      ;FOLD F324 = !E2164 & T8 + F324 ;%{SE}%MKUKATPVW %CVW_SPS %VBOASG %P 2:F324 = !E2164 & T8 + F324, 3: BOASG
         $FLAG[324] = NOT $IN[2164] AND $TIMER_FLAG[8] OR $FLAG[324]
      ;ENDFOLD
      ;FOLD -- RSK Sammelstoerung -- ;%{SE}%MKUKATPVW %CVW_COM %VCOMMENT %P 2:-- RSK Sammelstoerung --, 3: VW_COMMENT
      ;ENDFOLD
      ;FOLD F329 = F324 ;%{SE}%MKUKATPVW %CVW_SPS %VBOASG %P 2:F329 = F324, 3: BOASG
         $FLAG[329] = $FLAG[324]
      ;ENDFOLD
      ;FOLD A2164 = AUS ;%{SE}%MKUKATPVW %CVW_SPS %VBOASG %P 2:A2164 = AUS, 3: BOASG
         $OUT[2164] = FALSE
      ;ENDFOLD
      ;FOLD -- FRG Bewegung AUS -- ;%{SE}%MKUKATPVW %CVW_COM %VCOMMENT %P 2:-- FRG Bewegung AUS --, 3: VW_COMMENT
      ;ENDFOLD
      ;FOLD A2166 = AUS ;%{SE}%MKUKATPVW %CVW_SPS %VBOASG %P 2:A2166 = AUS, 3: BOASG
         $OUT[2166] = FALSE
      ;ENDFOLD
      ;FOLD -- FRG in Endlage halten ein -- ;%{SE}%MKUKATPVW %CVW_COM %VCOMMENT %P 2:-- FRG in Endlage halten ein --, 3: VW_COMMENT
      ;ENDFOLD
      ;FOLD A2165 = EIN ;%{SE}%MKUKATPVW %CVW_SPS %VBOASG %P 2:A2165 = EIN, 3: BOASG
         $OUT[2165] = TRUE
      ;ENDFOLD
      ;FOLD Schritt 154 = F324 & (E26 + E27) & A4039  ;%{SE}%MKUKATPVW %CVW_SPS %VST_CON %P 2:Schritt 154 = F324 & (E26 + E27) & A4039 , 3: ST_CON
         IF $FLAG[324] AND ($IN[26] OR $IN[27]) AND $OUT[4039] THEN
            PREVSTEP = $APP_INT[5]
            $APP_INT[5] = 154
         ENDIF
      ;ENDFOLD
      ;FOLD Schritt 158 = !F324 & E2164 & A4039  ;%{SE}%MKUKATPVW %CVW_SPS %VST_CON %P 2:Schritt 158 = !F324 & E2164 & A4039 , 3: ST_CON
         IF NOT $FLAG[324] AND $IN[2164] AND $OUT[4039] THEN
            PREVSTEP = $APP_INT[5]
            $APP_INT[5] = 158
         ENDIF
      ;ENDFOLD
   ;ENDFOLD
   ;FOLD SCHRITT 158 -- MS1 Reinigung (an Pneum. Schwenkeinheit MS1)-- ;%{P}%MKUKATPVW,%CSTEP,%VST_NR,%P 1:SCHRITT, 2:158, 3: MS1 Reinigung (an Pneum. Schwenkeinheit MS1)
      ;FOLD ;%{H}
         Case 158
      ;ENDFOLD
      ;FOLD -- Steuerluft EIN -- ;%{SE}%MKUKATPVW %CVW_COM %VCOMMENT %P 2:-- Steuerluft EIN --, 3: VW_COMMENT
      ;ENDFOLD
      ;FOLD A2161 = A4039 ;%{SE}%MKUKATPVW %CVW_SPS %VBOASG %P 2:A2161 = A4039, 3: BOASG
         $OUT[2161] = $OUT[4039]
      ;ENDFOLD
      ;FOLD A1864 = AUS ;%{SE}%MKUKATPVW %CVW_SPS %VBOASG %P 2:A1864 = AUS, 3: BOASG
         $OUT[1864] = FALSE
      ;ENDFOLD
      ;FOLD A2168 = AUS ;%{SE}%MKUKATPVW %CVW_SPS %VBOASG %P 2:A2168 = AUS, 3: BOASG
         $OUT[2168] = FALSE
      ;ENDFOLD
      ;FOLD -- Ueberwachungszeit Versetzeinheit/Brennerreinigung -- ;%{SE}%MKUKATPVW %CVW_COM %VCOMMENT %P 2:-- Ueberwachungszeit Versetzeinheit/Brennerreinigung --, 3: VW_COMMENT
      ;ENDFOLD
      ;FOLD t8 ( EIN ) = -100[1/10Sek] ;%{SE}%MKUKATPVW %CVW_SPS %VTASG %P 2:t8 ( EIN ) = -100[1/10Sek], 3: TASG
         VW(#SET_TIME,TRUE,8,0,-100)
      ;ENDFOLD
      ;FOLD Schritt 159 = A4039  ;%{SE}%MKUKATPVW %CVW_SPS %VST_CON %P 2:Schritt 159 = A4039 , 3: ST_CON
         IF $OUT[4039] THEN
            PREVSTEP = $APP_INT[5]
            $APP_INT[5] = 159
         ENDIF
      ;ENDFOLD
   ;ENDFOLD
   ;FOLD SCHRITT 159 -- MS1 Reinigung (an Pneum. Schwenkeinheit MS1)-- ;%{P}%MKUKATPVW,%CSTEP,%VST_NR,%P 1:SCHRITT, 2:159, 3: MS1 Reinigung (an Pneum. Schwenkeinheit MS1)
      ;FOLD ;%{H}
         Case 159
      ;ENDFOLD
      ;FOLD -- Steuerluft EIN -- ;%{SE}%MKUKATPVW %CVW_COM %VCOMMENT %P 2:-- Steuerluft EIN --, 3: VW_COMMENT
      ;ENDFOLD
      ;FOLD A2161 = A4039 ;%{SE}%MKUKATPVW %CVW_SPS %VBOASG %P 2:A2161 = A4039, 3: BOASG
         $OUT[2161] = $OUT[4039]
      ;ENDFOLD
      ;FOLD -- RSK Fehlerausgabe Versetzeinheit -- ;%{SE}%MKUKATPVW %CVW_COM %VCOMMENT %P 2:-- RSK Fehlerausgabe Versetzeinheit --, 3: VW_COMMENT
      ;ENDFOLD
      ;FOLD F328 = F576 & T8 ;%{SE}%MKUKATPVW %CVW_SPS %VBOASG %P 2:F328 = F576 & T8, 3: BOASG
         $FLAG[328] = $FLAG[576] AND $TIMER_FLAG[8]
      ;ENDFOLD
      ;FOLD -- RSK Sammelstoerung -- ;%{SE}%MKUKATPVW %CVW_COM %VCOMMENT %P 2:-- RSK Sammelstoerung --, 3: VW_COMMENT
      ;ENDFOLD
      ;FOLD F329 = T8 ;%{SE}%MKUKATPVW %CVW_SPS %VBOASG %P 2:F329 = T8, 3: BOASG
         $FLAG[329] = $TIMER_FLAG[8]
      ;ENDFOLD
      ;FOLD -- Versetzeinheit  in  Arbeitsst.  schw. -- ;%{SE}%MKUKATPVW %CVW_COM %VCOMMENT %P 2:-- Versetzeinheit  in  Arbeitsst.  schw. --, 3: VW_COMMENT
      ;ENDFOLD
      ;FOLD A2168 = !E2168 & E2164 & F576 ;%{SE}%MKUKATPVW %CVW_SPS %VBOASG %P 2:A2168 = !E2168 & E2164 & F576, 3: BOASG
         $OUT[2168] = NOT $IN[2168] AND $IN[2164] AND $FLAG[576]
      ;ENDFOLD
      ;FOLD Schritt 158 = A2168 & T8 & (E26 + E27) & A4039  ;%{SE}%MKUKATPVW %CVW_SPS %VST_CON %P 2:Schritt 158 = A2168 & T8 & (E26 + E27) & A4039 , 3: ST_CON
         IF $OUT[2168] AND $TIMER_FLAG[8] AND ($IN[26] OR $IN[27]) AND $OUT[4039] THEN
            PREVSTEP = $APP_INT[5]
            $APP_INT[5] = 158
         ENDIF
      ;ENDFOLD
      ;FOLD Schritt 160 = (E2168 & F576 + !E2168 & !F576) & A4039  ;%{SE}%MKUKATPVW %CVW_SPS %VST_CON %P 2:Schritt 160 = (E2168 & F576 + !E2168 & !F576) & A4039 , 3: ST_CON
         IF ($IN[2168] AND $FLAG[576] OR NOT $IN[2168] AND NOT $FLAG[576]) AND $OUT[4039] THEN
            PREVSTEP = $APP_INT[5]
            $APP_INT[5] = 160
         ENDIF
      ;ENDFOLD
   ;ENDFOLD
   ;FOLD SCHRITT 160 --MS1 Reinigung (an Pneum. Schwenkeinheit MS1)-- ;%{P}%MKUKATPVW,%CSTEP,%VST_NR,%P 1:SCHRITT, 2:160, 3:MS1 Reinigung (an Pneum. Schwenkeinheit MS1)
      ;FOLD ;%{H}
         Case 160
      ;ENDFOLD
      ;FOLD -- Steuerluft EIN -- ;%{SE}%MKUKATPVW %CVW_COM %VCOMMENT %P 2:-- Steuerluft EIN --, 3: VW_COMMENT
      ;ENDFOLD
      ;FOLD A2161 = A4039 ;%{SE}%MKUKATPVW %CVW_SPS %VBOASG %P 2:A2161 = A4039, 3: BOASG
         $OUT[2161] = $OUT[4039]
      ;ENDFOLD
      ;FOLD -- RSK Sammelstoerung -- ;%{SE}%MKUKATPVW %CVW_COM %VCOMMENT %P 2:-- RSK Sammelstoerung --, 3: VW_COMMENT
      ;ENDFOLD
      ;FOLD F329 = T8 ;%{SE}%MKUKATPVW %CVW_SPS %VBOASG %P 2:F329 = T8, 3: BOASG
         $FLAG[329] = $TIMER_FLAG[8]
      ;ENDFOLD
      ;FOLD -- Zeit Reinigung -- ;%{SE}%MKUKATPVW %CVW_COM %VCOMMENT %P 2:-- Zeit Reinigung --, 3: VW_COMMENT
      ;ENDFOLD
      ;FOLD F271 = i26 = 0 ;%{SE}%MKUKATPVW %CVW_SPS %VBOCMP %P 2:F271 = i26 = 0, 3: BOCMP
         $FLAG[271] = $COUNT_I[26] == 0
      ;ENDFOLD
      ;FOLD t9 ( F271 ) = -20[1/10Sek] ;%{SE}%MKUKATPVW %CVW_SPS %VTASG %P 2:t9 ( F271 ) = -20[1/10Sek], 3: TASG
         VW(#SET_TIME,$FLAG[271],9,0,-20)
      ;ENDFOLD
      ;FOLD t9 ( !F271 ) = i26[1/10Sek] ;%{SE}%MKUKATPVW %CVW_SPS %VTASG %P 2:t9 ( !F271 ) = i26[1/10Sek], 3: TASG
         VW(#SET_TIME,NOT $FLAG[271],9,0,$COUNT_I[26])
      ;ENDFOLD
      ;FOLD -- MS1 Ausblasen EIN -- ;%{SE}%MKUKATPVW %CVW_COM %VCOMMENT %P 2:-- MS1 Ausblasen EIN --, 3: VW_COMMENT
      ;ENDFOLD
      ;FOLD A1870 = EIN ;%{SE}%MKUKATPVW %CVW_SPS %VBOASG %P 2:A1870 = EIN, 3: BOASG
         $OUT[1870] = TRUE
      ;ENDFOLD
      ;FOLD -- MS1 Reinigung starten -- ;%{SE}%MKUKATPVW %CVW_COM %VCOMMENT %P 2:-- MS1 Reinigung starten --, 3: VW_COMMENT
      ;ENDFOLD
      ;FOLD A1864 = EIN ;%{SE}%MKUKATPVW %CVW_SPS %VBOASG %P 2:A1864 = EIN, 3: BOASG
         $OUT[1864] = TRUE
      ;ENDFOLD
      ;FOLD Schritt 158 = E1864 & T8 & (E26 + E27) & A4039  ;%{SE}%MKUKATPVW %CVW_SPS %VST_CON %P 2:Schritt 158 = E1864 & T8 & (E26 + E27) & A4039 , 3: ST_CON
         IF $IN[1864] AND $TIMER_FLAG[8] AND ($IN[26] OR $IN[27]) AND $OUT[4039] THEN
            PREVSTEP = $APP_INT[5]
            $APP_INT[5] = 158
         ENDIF
      ;ENDFOLD
      ;FOLD Schritt 161 = !E1864 & A4039  ;%{SE}%MKUKATPVW %CVW_SPS %VST_CON %P 2:Schritt 161 = !E1864 & A4039 , 3: ST_CON
         IF NOT $IN[1864] AND $OUT[4039] THEN
            PREVSTEP = $APP_INT[5]
            $APP_INT[5] = 161
         ENDIF
      ;ENDFOLD
   ;ENDFOLD
   ;FOLD SCHRITT 161 --MS1 Reinigung (an Pneum. Schwenkeinheit MS1)-- ;%{P}%MKUKATPVW,%CSTEP,%VST_NR,%P 1:SCHRITT, 2:161, 3:MS1 Reinigung (an Pneum. Schwenkeinheit MS1)
      ;FOLD ;%{H}
         Case 161
      ;ENDFOLD
      ;FOLD -- Steuerluft EIN -- ;%{SE}%MKUKATPVW %CVW_COM %VCOMMENT %P 2:-- Steuerluft EIN --, 3: VW_COMMENT
      ;ENDFOLD
      ;FOLD A2161 = A4039 ;%{SE}%MKUKATPVW %CVW_SPS %VBOASG %P 2:A2161 = A4039, 3: BOASG
         $OUT[2161] = $OUT[4039]
      ;ENDFOLD
      ;FOLD Schritt 158 = E1864 & T9 & (E26 + E27) & A4039  ;%{SE}%MKUKATPVW %CVW_SPS %VST_CON %P 2:Schritt 158 = E1864 & T9 & (E26 + E27) & A4039 , 3: ST_CON
         IF $IN[1864] AND $TIMER_FLAG[9] AND ($IN[26] OR $IN[27]) AND $OUT[4039] THEN
            PREVSTEP = $APP_INT[5]
            $APP_INT[5] = 158
         ENDIF
      ;ENDFOLD
      ;FOLD Schritt 162 = T9 & A4039  ;%{SE}%MKUKATPVW %CVW_SPS %VST_CON %P 2:Schritt 162 = T9 & A4039 , 3: ST_CON
         IF $TIMER_FLAG[9] AND $OUT[4039] THEN
            PREVSTEP = $APP_INT[5]
            $APP_INT[5] = 162
         ENDIF
      ;ENDFOLD
   ;ENDFOLD
   ;FOLD SCHRITT 162 --MS1 Reinigung (an Pneum. Schwenkeinheit MS1)-- ;%{P}%MKUKATPVW,%CSTEP,%VST_NR,%P 1:SCHRITT, 2:162, 3:MS1 Reinigung (an Pneum. Schwenkeinheit MS1)
      ;FOLD ;%{H}
         Case 162
      ;ENDFOLD
      ;FOLD -- Steuerluft EIN -- ;%{SE}%MKUKATPVW %CVW_COM %VCOMMENT %P 2:-- Steuerluft EIN --, 3: VW_COMMENT
      ;ENDFOLD
      ;FOLD A2161 = A4039 ;%{SE}%MKUKATPVW %CVW_SPS %VBOASG %P 2:A2161 = A4039, 3: BOASG
         $OUT[2161] = $OUT[4039]
      ;ENDFOLD
      ;FOLD -- RSK Sammelstoerung -- ;%{SE}%MKUKATPVW %CVW_COM %VCOMMENT %P 2:-- RSK Sammelstoerung --, 3: VW_COMMENT
      ;ENDFOLD
      ;FOLD F329 = T8 ;%{SE}%MKUKATPVW %CVW_SPS %VBOASG %P 2:F329 = T8, 3: BOASG
         $FLAG[329] = $TIMER_FLAG[8]
      ;ENDFOLD
      ;FOLD -- MS1 Reinigung beenden -- ;%{SE}%MKUKATPVW %CVW_COM %VCOMMENT %P 2:-- MS1 Reinigung beenden --, 3: VW_COMMENT
      ;ENDFOLD
      ;FOLD A1864 = AUS ;%{SE}%MKUKATPVW %CVW_SPS %VBOASG %P 2:A1864 = AUS, 3: BOASG
         $OUT[1864] = FALSE
      ;ENDFOLD
      ;FOLD -- MS1 Ausblasen AUS -- ;%{SE}%MKUKATPVW %CVW_COM %VCOMMENT %P 2:-- MS1 Ausblasen AUS --, 3: VW_COMMENT
      ;ENDFOLD
      ;FOLD A1870 = AUS ;%{SE}%MKUKATPVW %CVW_SPS %VBOASG %P 2:A1870 = AUS, 3: BOASG
         $OUT[1870] = FALSE
      ;ENDFOLD
      ;FOLD -- MS1 Einspruehen EIN -- ;%{SE}%MKUKATPVW %CVW_COM %VCOMMENT %P 2:-- MS1 Einspruehen EIN --, 3: VW_COMMENT
      ;ENDFOLD
      ;FOLD A520 = !F574 & F575 ;%{SE}%MKUKATPVW %CVW_SPS %VBOASG %P 2:A520 = !F574 & F575, 3: BOASG
         $OUT[520] = NOT $FLAG[574] AND $FLAG[575]
      ;ENDFOLD
      ;FOLD A1871 = F574 & F575 ;%{SE}%MKUKATPVW %CVW_SPS %VBOASG %P 2:A1871 = F574 & F575, 3: BOASG
         $OUT[1871] = $FLAG[574] AND $FLAG[575]
      ;ENDFOLD
      ;FOLD -- Einschaltdauer Einspruehen -- ;%{SE}%MKUKATPVW %CVW_COM %VCOMMENT %P 2:-- Einschaltdauer Einspruehen --, 3: VW_COMMENT
      ;ENDFOLD
      ;FOLD t7 ( EIN ) = i23[1/10Sek] ;%{SE}%MKUKATPVW %CVW_SPS %VTASG %P 2:t7 ( EIN ) = i23[1/10Sek], 3: TASG
         VW(#SET_TIME,TRUE,7,0,$COUNT_I[23])
      ;ENDFOLD
      ;FOLD Schritt 163 = E1864 & A4039  ;%{SE}%MKUKATPVW %CVW_SPS %VST_CON %P 2:Schritt 163 = E1864 & A4039 , 3: ST_CON
         IF $IN[1864] AND $OUT[4039] THEN
            PREVSTEP = $APP_INT[5]
            $APP_INT[5] = 163
         ENDIF
      ;ENDFOLD
   ;ENDFOLD
   ;FOLD SCHRITT 163 --MS1 Reinigung (an Pneum. Schwenkeinheit MS1)-- ;%{P}%MKUKATPVW,%CSTEP,%VST_NR,%P 1:SCHRITT, 2:163, 3:MS1 Reinigung (an Pneum. Schwenkeinheit MS1)
      ;FOLD ;%{H}
         Case 163
      ;ENDFOLD
      ;FOLD F323 = AUS ;%{SE}%MKUKATPVW %CVW_SPS %VBOASG %P 2:F323 = AUS, 3: BOASG
         $FLAG[323] = FALSE
      ;ENDFOLD
      ;FOLD A2163 = AUS ;%{SE}%MKUKATPVW %CVW_SPS %VBOASG %P 2:A2163 = AUS, 3: BOASG
         $OUT[2163] = FALSE
      ;ENDFOLD
      ;FOLD A2164 = AUS ;%{SE}%MKUKATPVW %CVW_SPS %VBOASG %P 2:A2164 = AUS, 3: BOASG
         $OUT[2164] = FALSE
      ;ENDFOLD
      ;FOLD A2165 = AUS ;%{SE}%MKUKATPVW %CVW_SPS %VBOASG %P 2:A2165 = AUS, 3: BOASG
         $OUT[2165] = FALSE
      ;ENDFOLD
      ;FOLD A2166 = AUS ;%{SE}%MKUKATPVW %CVW_SPS %VBOASG %P 2:A2166 = AUS, 3: BOASG
         $OUT[2166] = FALSE
      ;ENDFOLD
      ;FOLD A2168 = AUS ;%{SE}%MKUKATPVW %CVW_SPS %VBOASG %P 2:A2168 = AUS, 3: BOASG
         $OUT[2168] = FALSE
      ;ENDFOLD
      ;FOLD -- Ueberwachungszeit Schwenkeinheit 1 schwenken -- ;%{SE}%MKUKATPVW %CVW_COM %VCOMMENT %P 2:-- Ueberwachungszeit Schwenkeinheit 1 schwenken --, 3: VW_COMMENT
      ;ENDFOLD
      ;FOLD t8 ( EIN ) = -100[1/10Sek] ;%{SE}%MKUKATPVW %CVW_SPS %VTASG %P 2:t8 ( EIN ) = -100[1/10Sek], 3: TASG
         VW(#SET_TIME,TRUE,8,0,-100)
      ;ENDFOLD
      ;FOLD Schritt 164 = T7 & A4039  ;%{SE}%MKUKATPVW %CVW_SPS %VST_CON %P 2:Schritt 164 = T7 & A4039 , 3: ST_CON
         IF $TIMER_FLAG[7] AND $OUT[4039] THEN
            PREVSTEP = $APP_INT[5]
            $APP_INT[5] = 164
         ENDIF
      ;ENDFOLD
   ;ENDFOLD
   ;FOLD SCHRITT 164 --MS1 Reinigung (an Pneum. Schwenkeinheit MS1)-- ;%{P}%MKUKATPVW,%CSTEP,%VST_NR,%P 1:SCHRITT, 2:164, 3:MS1 Reinigung (an Pneum. Schwenkeinheit MS1)
      ;FOLD ;%{H}
         Case 164
      ;ENDFOLD
      ;FOLD -- Steuerluft EIN -- ;%{SE}%MKUKATPVW %CVW_COM %VCOMMENT %P 2:-- Steuerluft EIN --, 3: VW_COMMENT
      ;ENDFOLD
      ;FOLD A2161 = A4039 ;%{SE}%MKUKATPVW %CVW_SPS %VBOASG %P 2:A2161 = A4039, 3: BOASG
         $OUT[2161] = $OUT[4039]
      ;ENDFOLD
      ;FOLD -- MS1 Einspruehen AUS -- ;%{SE}%MKUKATPVW %CVW_COM %VCOMMENT %P 2:-- MS1 Einspruehen AUS --, 3: VW_COMMENT
      ;ENDFOLD
      ;FOLD A520 = AUS ;%{SE}%MKUKATPVW %CVW_SPS %VBOASG %P 2:A520 = AUS, 3: BOASG
         $OUT[520] = FALSE
      ;ENDFOLD
      ;FOLD A1871 = AUS ;%{SE}%MKUKATPVW %CVW_SPS %VBOASG %P 2:A1871 = AUS, 3: BOASG
         $OUT[1871] = FALSE
      ;ENDFOLD
      ;FOLD -- Versetzeinheit in Ruhest. schw. -- ;%{SE}%MKUKATPVW %CVW_COM %VCOMMENT %P 2:-- Versetzeinheit in Ruhest. schw. --, 3: VW_COMMENT
      ;ENDFOLD
      ;FOLD A2167 = EIN ;%{SE}%MKUKATPVW %CVW_SPS %VBOASG %P 2:A2167 = EIN, 3: BOASG
         $OUT[2167] = TRUE
      ;ENDFOLD
      ;FOLD A2168 = AUS ;%{SE}%MKUKATPVW %CVW_SPS %VBOASG %P 2:A2168 = AUS, 3: BOASG
         $OUT[2168] = FALSE
      ;ENDFOLD
      ;FOLD -- RSK Fehlerausgabe Versetzeinheit in Ruhest. schw. -- ;%{SE}%MKUKATPVW %CVW_COM %VCOMMENT %P 2:-- RSK Fehlerausgabe Versetzeinheit in Ruhest. schw. --, 3: VW_COMMENT
      ;ENDFOLD
      ;FOLD F328 = F576 & T8 ;%{SE}%MKUKATPVW %CVW_SPS %VBOASG %P 2:F328 = F576 & T8, 3: BOASG
         $FLAG[328] = $FLAG[576] AND $TIMER_FLAG[8]
      ;ENDFOLD
      ;FOLD -- RSK Fehlerausgabe Schwenkeinheit 1 Arbeit. -- ;%{SE}%MKUKATPVW %CVW_COM %VCOMMENT %P 2:-- RSK Fehlerausgabe Schwenkeinheit 1 Arbeit. --, 3: VW_COMMENT
      ;ENDFOLD
      ;FOLD F324 = !E2164 & T8 ;%{SE}%MKUKATPVW %CVW_SPS %VBOASG %P 2:F324 = !E2164 & T8, 3: BOASG
         $FLAG[324] = NOT $IN[2164] AND $TIMER_FLAG[8]
      ;ENDFOLD
      ;FOLD -- RSK Sammelstoerung -- ;%{SE}%MKUKATPVW %CVW_COM %VCOMMENT %P 2:-- RSK Sammelstoerung --, 3: VW_COMMENT
      ;ENDFOLD
      ;FOLD F329 = F324 + F328 ;%{SE}%MKUKATPVW %CVW_SPS %VBOASG %P 2:F329 = F324 + F328, 3: BOASG
         $FLAG[329] = $FLAG[324] OR $FLAG[328]
      ;ENDFOLD
      ;FOLD Schritt 163 = (E26 + E27) & (F324 + F328) & A4039  ;%{SE}%MKUKATPVW %CVW_SPS %VST_CON %P 2:Schritt 163 = (E26 + E27) & (F324 + F328) & A4039 , 3: ST_CON
         IF ($IN[26] OR $IN[27]) AND ($FLAG[324] OR $FLAG[328]) AND $OUT[4039] THEN
            PREVSTEP = $APP_INT[5]
            $APP_INT[5] = 163
         ENDIF
      ;ENDFOLD
      ;FOLD Schritt 165 = (!F324 + T8) & (F523 & !F524 & E2161 + !F523 & F524 & !E2162) & E2167 & F576 & A4039  ;%{SE}%MKUKATPVW %CVW_SPS %VST_CON %P 2:Schritt 165 = (!F324 + T8) & (F523 & !F524 & E2161 + !F523 & F524 & !E2162) & E2167 & F576 & A4039 , 3: ST_CON
         IF (NOT $FLAG[324] OR $TIMER_FLAG[8]) AND ($FLAG[523] AND NOT $FLAG[524] AND $IN[2161] OR NOT $FLAG[523] AND $FLAG[524] AND NOT $IN[2162]) AND $IN[2167] AND $FLAG[576] AND $OUT[4039] THEN
            PREVSTEP = $APP_INT[5]
            $APP_INT[5] = 165
         ENDIF
      ;ENDFOLD
      ;FOLD Schritt 165 = (!F324 + T8) & (F523 & !F524 & E2161 + !F523 & F524 & !E2162) & !E2167 & !F576 & A4039  ;%{SE}%MKUKATPVW %CVW_SPS %VST_CON %P 2:Schritt 165 = (!F324 + T8) & (F523 & !F524 & E2161 + !F523 & F524 & !E2162) & !E2167 & !F576 & A4039 , 3: ST_CON
         IF (NOT $FLAG[324] OR $TIMER_FLAG[8]) AND ($FLAG[523] AND NOT $FLAG[524] AND $IN[2161] OR NOT $FLAG[523] AND $FLAG[524] AND NOT $IN[2162]) AND NOT $IN[2167] AND NOT $FLAG[576] AND $OUT[4039] THEN
            PREVSTEP = $APP_INT[5]
            $APP_INT[5] = 165
         ENDIF
      ;ENDFOLD
   ;ENDFOLD
   ;FOLD SCHRITT 165 --MS1 Reinigung (an Pneum. Schwenkeinheit MS1)-- ;%{P}%MKUKATPVW,%CSTEP,%VST_NR,%P 1:SCHRITT, 2:165, 3:MS1 Reinigung (an Pneum. Schwenkeinheit MS1)
      ;FOLD ;%{H}
         Case 165
      ;ENDFOLD
      ;FOLD -- Steuerluft EIN -- ;%{SE}%MKUKATPVW %CVW_COM %VCOMMENT %P 2:-- Steuerluft EIN --, 3: VW_COMMENT
      ;ENDFOLD
      ;FOLD A2161 = A4039 ;%{SE}%MKUKATPVW %CVW_SPS %VBOASG %P 2:A2161 = A4039, 3: BOASG
         $OUT[2161] = $OUT[4039]
      ;ENDFOLD
      ;FOLD A2167 = AUS ;%{SE}%MKUKATPVW %CVW_SPS %VBOASG %P 2:A2167 = AUS, 3: BOASG
         $OUT[2167] = FALSE
      ;ENDFOLD
      ;FOLD -- Schwenkeinheit 1 in Ruhestellung schwenken -- ;%{SE}%MKUKATPVW %CVW_COM %VCOMMENT %P 2:-- Schwenkeinheit 1 in Ruhestellung schwenken --, 3: VW_COMMENT
      ;ENDFOLD
      ;FOLD A2163 = !E2163 ;%{SE}%MKUKATPVW %CVW_SPS %VBOASG %P 2:A2163 = !E2163, 3: BOASG
         $OUT[2163] = NOT $IN[2163]
      ;ENDFOLD
      ;FOLD A2164 = AUS ;%{SE}%MKUKATPVW %CVW_SPS %VBOASG %P 2:A2164 = AUS, 3: BOASG
         $OUT[2164] = FALSE
      ;ENDFOLD
      ;FOLD -- FRG Bewegung EIN -- ;%{SE}%MKUKATPVW %CVW_COM %VCOMMENT %P 2:-- FRG Bewegung EIN --, 3: VW_COMMENT
      ;ENDFOLD
      ;FOLD A2165 = AUS ;%{SE}%MKUKATPVW %CVW_SPS %VBOASG %P 2:A2165 = AUS, 3: BOASG
         $OUT[2165] = FALSE
      ;ENDFOLD
      ;FOLD A2166 = !E2163 ;%{SE}%MKUKATPVW %CVW_SPS %VBOASG %P 2:A2166 = !E2163, 3: BOASG
         $OUT[2166] = NOT $IN[2163]
      ;ENDFOLD
      ;FOLD Schritt 166 = E1864 & !E2164 & E2163 & A4039 + T8  ;%{SE}%MKUKATPVW %CVW_SPS %VST_CON %P 2:Schritt 166 = E1864 & !E2164 & E2163 & A4039 + T8 , 3: ST_CON
         IF $IN[1864] AND NOT $IN[2164] AND $IN[2163] AND $OUT[4039] OR $TIMER_FLAG[8] THEN
            PREVSTEP = $APP_INT[5]
            $APP_INT[5] = 166
         ENDIF
      ;ENDFOLD
   ;ENDFOLD
   ;FOLD SCHRITT 166 --MS1 Reinigung (an Pneum. Schwenkeinheit MS1)-- ;%{P}%MKUKATPVW,%CSTEP,%VST_NR,%P 1:SCHRITT, 2:166, 3:MS1 Reinigung (an Pneum. Schwenkeinheit MS1)
      ;FOLD ;%{H}
         Case 166
      ;ENDFOLD
      ;FOLD -- Steuerluft EIN -- ;%{SE}%MKUKATPVW %CVW_COM %VCOMMENT %P 2:-- Steuerluft EIN --, 3: VW_COMMENT
      ;ENDFOLD
      ;FOLD A2161 = A4039 ;%{SE}%MKUKATPVW %CVW_SPS %VBOASG %P 2:A2161 = A4039, 3: BOASG
         $OUT[2161] = $OUT[4039]
      ;ENDFOLD
      ;FOLD -- RSK Fehlerausgabe Schwenkeinheit 1 Ruhestellung -- ;%{SE}%MKUKATPVW %CVW_COM %VCOMMENT %P 2:-- RSK Fehlerausgabe Schwenkeinheit 1 Ruhestellung --, 3: VW_COMMENT
      ;ENDFOLD
      ;FOLD F323 = !E2163 & T8 + F323 ;%{SE}%MKUKATPVW %CVW_SPS %VBOASG %P 2:F323 = !E2163 & T8 + F323, 3: BOASG
         $FLAG[323] = NOT $IN[2163] AND $TIMER_FLAG[8] OR $FLAG[323]
      ;ENDFOLD
      ;FOLD -- RSK Sammelstoerung -- ;%{SE}%MKUKATPVW %CVW_COM %VCOMMENT %P 2:-- RSK Sammelstoerung --, 3: VW_COMMENT
      ;ENDFOLD
      ;FOLD F329 = F323 ;%{SE}%MKUKATPVW %CVW_SPS %VBOASG %P 2:F329 = F323, 3: BOASG
         $FLAG[329] = $FLAG[323]
      ;ENDFOLD
      ;FOLD A2163 = AUS ;%{SE}%MKUKATPVW %CVW_SPS %VBOASG %P 2:A2163 = AUS, 3: BOASG
         $OUT[2163] = FALSE
      ;ENDFOLD
      ;FOLD -- FRG Bewegung AUS -- ;%{SE}%MKUKATPVW %CVW_COM %VCOMMENT %P 2:-- FRG Bewegung AUS --, 3: VW_COMMENT
      ;ENDFOLD
      ;FOLD A2166 = AUS ;%{SE}%MKUKATPVW %CVW_SPS %VBOASG %P 2:A2166 = AUS, 3: BOASG
         $OUT[2166] = FALSE
      ;ENDFOLD
      ;FOLD Schritt 163 = F323 & (E26 + E27) & A4039  ;%{SE}%MKUKATPVW %CVW_SPS %VST_CON %P 2:Schritt 163 = F323 & (E26 + E27) & A4039 , 3: ST_CON
         IF $FLAG[323] AND ($IN[26] OR $IN[27]) AND $OUT[4039] THEN
            PREVSTEP = $APP_INT[5]
            $APP_INT[5] = 163
         ENDIF
      ;ENDFOLD
      ;FOLD Schritt 167 = !F323 & (E2166 + F837) & A4039  ;%{SE}%MKUKATPVW %CVW_SPS %VST_CON %P 2:Schritt 167 = !F323 & (E2166 + F837) & A4039 , 3: ST_CON
         IF NOT $FLAG[323] AND ($IN[2166] OR $FLAG[837]) AND $OUT[4039] THEN
            PREVSTEP = $APP_INT[5]
            $APP_INT[5] = 167
         ENDIF
      ;ENDFOLD
   ;ENDFOLD
   ;FOLD SCHRITT 167 --MS1 Reinigung (an Pneum. Schwenkeinheit MS1)-- ;%{P}%MKUKATPVW,%CSTEP,%VST_NR,%P 1:SCHRITT, 2:167, 3:MS1 Reinigung (an Pneum. Schwenkeinheit MS1)
      ;FOLD ;%{H}
         Case 167
      ;ENDFOLD
      ;FOLD -- Steuerluft EIN -- ;%{SE}%MKUKATPVW %CVW_COM %VCOMMENT %P 2:-- Steuerluft EIN --, 3: VW_COMMENT
      ;ENDFOLD
      ;FOLD A2161 = A4039 ;%{SE}%MKUKATPVW %CVW_SPS %VBOASG %P 2:A2161 = A4039, 3: BOASG
         $OUT[2161] = $OUT[4039]
      ;ENDFOLD
      ;FOLD -- RSK Sammelstoerung -- ;%{SE}%MKUKATPVW %CVW_COM %VCOMMENT %P 2:-- RSK Sammelstoerung --, 3: VW_COMMENT
      ;ENDFOLD
      ;FOLD F329 = T8 ;%{SE}%MKUKATPVW %CVW_SPS %VBOASG %P 2:F329 = T8, 3: BOASG
         $FLAG[329] = $TIMER_FLAG[8]
      ;ENDFOLD
      ;FOLD F323 = AUS ;%{SE}%MKUKATPVW %CVW_SPS %VBOASG %P 2:F323 = AUS, 3: BOASG
         $FLAG[323] = FALSE
      ;ENDFOLD
      ;FOLD -- FRG in Endlage halten ein -- ;%{SE}%MKUKATPVW %CVW_COM %VCOMMENT %P 2:-- FRG in Endlage halten ein --, 3: VW_COMMENT
      ;ENDFOLD
      ;FOLD A2165 = EIN ;%{SE}%MKUKATPVW %CVW_SPS %VBOASG %P 2:A2165 = EIN, 3: BOASG
         $OUT[2165] = TRUE
      ;ENDFOLD
      ;FOLD Schritt 168 = !E2165 & (E2166 + F837) & A4039  ;%{SE}%MKUKATPVW %CVW_SPS %VST_CON %P 2:Schritt 168 = !E2165 & (E2166 + F837) & A4039 , 3: ST_CON
         IF NOT $IN[2165] AND ($IN[2166] OR $FLAG[837]) AND $OUT[4039] THEN
            PREVSTEP = $APP_INT[5]
            $APP_INT[5] = 168
         ENDIF
      ;ENDFOLD
   ;ENDFOLD
   ;FOLD SCHRITT 168 --MS1 Reinigung (an Pneum. Schwenkeinheit MS1)-- ;%{P}%MKUKATPVW,%CSTEP,%VST_NR,%P 1:SCHRITT, 2:168, 3:MS1 Reinigung (an Pneum. Schwenkeinheit MS1)
      ;FOLD ;%{H}
         Case 168
      ;ENDFOLD
      ;FOLD -- Steuerluft EIN -- ;%{SE}%MKUKATPVW %CVW_COM %VCOMMENT %P 2:-- Steuerluft EIN --, 3: VW_COMMENT
      ;ENDFOLD
      ;FOLD A2161 = A4039 ;%{SE}%MKUKATPVW %CVW_SPS %VBOASG %P 2:A2161 = A4039, 3: BOASG
         $OUT[2161] = $OUT[4039]
      ;ENDFOLD
      ;FOLD -- FRG in Endlage halten AUS -- ;%{SE}%MKUKATPVW %CVW_COM %VCOMMENT %P 2:-- FRG in Endlage halten AUS --, 3: VW_COMMENT
      ;ENDFOLD
      ;FOLD A2165 = AUS ;%{SE}%MKUKATPVW %CVW_SPS %VBOASG %P 2:A2165 = AUS, 3: BOASG
         $OUT[2165] = FALSE
      ;ENDFOLD
      ;FOLD -- MS1 Zaehler ruecksetzen -- ;%{SE}%MKUKATPVW %CVW_COM %VCOMMENT %P 2:-- MS1 Zaehler ruecksetzen --, 3: VW_COMMENT
      ;ENDFOLD
      ;FOLD -- MS1 FRG Reinigung -- ;%{SE}%MKUKATPVW %CVW_COM %VCOMMENT %P 2:-- MS1 FRG Reinigung --, 3: VW_COMMENT
      ;ENDFOLD
      ;FOLD F603 = AUS ;%{SE}%MKUKATPVW %CVW_SPS %VBOASG %P 2:F603 = AUS, 3: BOASG
         $FLAG[603] = FALSE
      ;ENDFOLD
      ;FOLD -- MS1 Reinigung FK -- ;%{SE}%MKUKATPVW %CVW_COM %VCOMMENT %P 2:-- MS1 Reinigung FK --, 3: VW_COMMENT
      ;ENDFOLD
      ;FOLD F605 = EIN ;%{SE}%MKUKATPVW %CVW_SPS %VBOASG %P 2:F605 = EIN, 3: BOASG
         $FLAG[605] = TRUE
      ;ENDFOLD
      ;FOLD t8 ( EIN ) = STOP ;%{SE}%MKUKATPVW %CVW_SPS %VTSTOP %P 2:t8 ( EIN ) = STOP, 3: TSTOP
         VW(#SET_TIME,TRUE,8,1,0)
      ;ENDFOLD
      ;FOLD Schritt 1 = A4039  ;%{SE}%MKUKATPVW %CVW_SPS %VST_CON %P 2:Schritt 1 = A4039 , 3: ST_CON
         IF $OUT[4039] THEN
            PREVSTEP = $APP_INT[5]
            $APP_INT[5] = 1
         ENDIF
      ;ENDFOLD
   ;ENDFOLD
   ;FOLD SCHRITT 169 --MS2 Reinigung (an Pneum. Schwenkeinheit MS2)-- ;%{P}%MKUKATPVW,%CSTEP,%VST_NR,%P 1:SCHRITT, 2:169, 3:MS2 Reinigung (an Pneum. Schwenkeinheit MS2)
      ;FOLD ;%{H}
         Case 169
      ;ENDFOLD
      ;FOLD -- RSK gestartet -- ;%{SE}%MKUKATPVW %CVW_COM %VCOMMENT %P 2:-- RSK gestartet --, 3: VW_COMMENT
      ;ENDFOLD
      ;FOLD F321 = AUS ;%{SE}%MKUKATPVW %CVW_SPS %VBOASG %P 2:F321 = AUS, 3: BOASG
         $FLAG[321] = FALSE
      ;ENDFOLD
      ;FOLD F323 = AUS ;%{SE}%MKUKATPVW %CVW_SPS %VBOASG %P 2:F323 = AUS, 3: BOASG
         $FLAG[323] = FALSE
      ;ENDFOLD
      ;FOLD F324 = AUS ;%{SE}%MKUKATPVW %CVW_SPS %VBOASG %P 2:F324 = AUS, 3: BOASG
         $FLAG[324] = FALSE
      ;ENDFOLD
      ;FOLD F329 = AUS ;%{SE}%MKUKATPVW %CVW_SPS %VBOASG %P 2:F329 = AUS, 3: BOASG
         $FLAG[329] = FALSE
      ;ENDFOLD
      ;FOLD -- MS2 Reinigung gestartet -- ;%{SE}%MKUKATPVW %CVW_COM %VCOMMENT %P 2:-- MS2 Reinigung gestartet --, 3: VW_COMMENT
      ;ENDFOLD
      ;FOLD F608 = EIN ;%{SE}%MKUKATPVW %CVW_SPS %VBOASG %P 2:F608 = EIN, 3: BOASG
         $FLAG[608] = TRUE
      ;ENDFOLD
      ;FOLD -- MS bei Reinigung -- ;%{SE}%MKUKATPVW %CVW_COM %VCOMMENT %P 2:-- MS bei Reinigung --, 3: VW_COMMENT
      ;ENDFOLD
      ;FOLD A116 = EIN ;%{SE}%MKUKATPVW %CVW_SPS %VBOASG %P 2:A116 = EIN, 3: BOASG
         $OUT[116] = TRUE
      ;ENDFOLD
      ;FOLD -- Steuerluft EIN -- ;%{SE}%MKUKATPVW %CVW_COM %VCOMMENT %P 2:-- Steuerluft EIN --, 3: VW_COMMENT
      ;ENDFOLD
      ;FOLD A2169 = A4039 ;%{SE}%MKUKATPVW %CVW_SPS %VBOASG %P 2:A2169 = A4039, 3: BOASG
         $OUT[2169] = $OUT[4039]
      ;ENDFOLD
      ;FOLD A2171 = AUS ;%{SE}%MKUKATPVW %CVW_SPS %VBOASG %P 2:A2171 = AUS, 3: BOASG
         $OUT[2171] = FALSE
      ;ENDFOLD
      ;FOLD A2172 = AUS ;%{SE}%MKUKATPVW %CVW_SPS %VBOASG %P 2:A2172 = AUS, 3: BOASG
         $OUT[2172] = FALSE
      ;ENDFOLD
      ;FOLD A2173 = AUS ;%{SE}%MKUKATPVW %CVW_SPS %VBOASG %P 2:A2173 = AUS, 3: BOASG
         $OUT[2173] = FALSE
      ;ENDFOLD
      ;FOLD A2174 = AUS ;%{SE}%MKUKATPVW %CVW_SPS %VBOASG %P 2:A2174 = AUS, 3: BOASG
         $OUT[2174] = FALSE
      ;ENDFOLD
      ;FOLD A2175 = AUS ;%{SE}%MKUKATPVW %CVW_SPS %VBOASG %P 2:A2175 = AUS, 3: BOASG
         $OUT[2175] = FALSE
      ;ENDFOLD
      ;FOLD A2176 = AUS ;%{SE}%MKUKATPVW %CVW_SPS %VBOASG %P 2:A2176 = AUS, 3: BOASG
         $OUT[2176] = FALSE
      ;ENDFOLD
      ;FOLD -- Ueberwachungszeit Schwenkeinheit 2 -- ;%{SE}%MKUKATPVW %CVW_COM %VCOMMENT %P 2:-- Ueberwachungszeit Schwenkeinheit 2 --, 3: VW_COMMENT
      ;ENDFOLD
      ;FOLD t8 ( EIN ) = -100[1/10Sek] ;%{SE}%MKUKATPVW %CVW_SPS %VTASG %P 2:t8 ( EIN ) = -100[1/10Sek], 3: TASG
         VW(#SET_TIME,TRUE,8,0,-100)
      ;ENDFOLD
      ;FOLD Schritt 170 = A4039  ;%{SE}%MKUKATPVW %CVW_SPS %VST_CON %P 2:Schritt 170 = A4039 , 3: ST_CON
         IF $OUT[4039] THEN
            PREVSTEP = $APP_INT[5]
            $APP_INT[5] = 170
         ENDIF
      ;ENDFOLD
   ;ENDFOLD
   ;FOLD SCHRITT 170 --MS2 Reinigung (an Pneum. Schwenkeinheit MS2)-- ;%{P}%MKUKATPVW,%CSTEP,%VST_NR,%P 1:SCHRITT, 2:170, 3:MS2 Reinigung (an Pneum. Schwenkeinheit MS2)
      ;FOLD ;%{H}
         Case 170
      ;ENDFOLD
      ;FOLD -- Steuerluft EIN -- ;%{SE}%MKUKATPVW %CVW_COM %VCOMMENT %P 2:-- Steuerluft EIN --, 3: VW_COMMENT
      ;ENDFOLD
      ;FOLD A2169 = A4039 ;%{SE}%MKUKATPVW %CVW_SPS %VBOASG %P 2:A2169 = A4039, 3: BOASG
         $OUT[2169] = $OUT[4039]
      ;ENDFOLD
      ;FOLD -- RSK Fehlerausgabe Schwenkeinheit 2 Ruhest. -- ;%{SE}%MKUKATPVW %CVW_COM %VCOMMENT %P 2:-- RSK Fehlerausgabe Schwenkeinheit 2 Ruhest. --, 3: VW_COMMENT
      ;ENDFOLD
      ;FOLD F323 = !E2171 & T8 ;%{SE}%MKUKATPVW %CVW_SPS %VBOASG %P 2:F323 = !E2171 & T8, 3: BOASG
         $FLAG[323] = NOT $IN[2171] AND $TIMER_FLAG[8]
      ;ENDFOLD
      ;FOLD -- RSK Sammelstoerung -- ;%{SE}%MKUKATPVW %CVW_COM %VCOMMENT %P 2:-- RSK Sammelstoerung --, 3: VW_COMMENT
      ;ENDFOLD
      ;FOLD F329 = F323 + T8 ;%{SE}%MKUKATPVW %CVW_SPS %VBOASG %P 2:F329 = F323 + T8, 3: BOASG
         $FLAG[329] = $FLAG[323] OR $TIMER_FLAG[8]
      ;ENDFOLD
      ;FOLD Schritt 169 = (E26 + E27) & F323 & A4039  ;%{SE}%MKUKATPVW %CVW_SPS %VST_CON %P 2:Schritt 169 = (E26 + E27) & F323 & A4039 , 3: ST_CON
         IF ($IN[26] OR $IN[27]) AND $FLAG[323] AND $OUT[4039] THEN
            PREVSTEP = $APP_INT[5]
            $APP_INT[5] = 169
         ENDIF
      ;ENDFOLD
      ;FOLD Schritt 171 = (!F323 + T8) & (F523 & !F524 & E2169 + !F523 & F524 & !E2170) & A4039  ;%{SE}%MKUKATPVW %CVW_SPS %VST_CON %P 2:Schritt 171 = (!F323 + T8) & (F523 & !F524 & E2169 + !F523 & F524 & !E2170) & A4039 , 3: ST_CON
         IF (NOT $FLAG[323] OR $TIMER_FLAG[8]) AND ($FLAG[523] AND NOT $FLAG[524] AND $IN[2169] OR NOT $FLAG[523] AND $FLAG[524] AND NOT $IN[2170]) AND $OUT[4039] THEN
            PREVSTEP = $APP_INT[5]
            $APP_INT[5] = 171
         ENDIF
      ;ENDFOLD
   ;ENDFOLD
   ;FOLD SCHRITT 171 --MS2 Reinigung (an Pneum. Schwenkeinheit MS2)-- ;%{P}%MKUKATPVW,%CSTEP,%VST_NR,%P 1:SCHRITT, 2:171, 3:MS2 Reinigung (an Pneum. Schwenkeinheit MS2)
      ;FOLD ;%{H}
         Case 171
      ;ENDFOLD
      ;FOLD -- Steuerluft EIN -- ;%{SE}%MKUKATPVW %CVW_COM %VCOMMENT %P 2:-- Steuerluft EIN --, 3: VW_COMMENT
      ;ENDFOLD
      ;FOLD A2169 = A4039 ;%{SE}%MKUKATPVW %CVW_SPS %VBOASG %P 2:A2169 = A4039, 3: BOASG
         $OUT[2169] = $OUT[4039]
      ;ENDFOLD
      ;FOLD -- Schwenkeinheit 2 in Arbeitsstellung schwenken -- ;%{SE}%MKUKATPVW %CVW_COM %VCOMMENT %P 2:-- Schwenkeinheit 2 in Arbeitsstellung schwenken --, 3: VW_COMMENT
      ;ENDFOLD
      ;FOLD A2172 = EIN ;%{SE}%MKUKATPVW %CVW_SPS %VBOASG %P 2:A2172 = EIN, 3: BOASG
         $OUT[2172] = TRUE
      ;ENDFOLD
      ;FOLD -- FRG Bewegung EIN -- ;%{SE}%MKUKATPVW %CVW_COM %VCOMMENT %P 2:-- FRG Bewegung EIN --, 3: VW_COMMENT
      ;ENDFOLD
      ;FOLD A2173 = AUS ;%{SE}%MKUKATPVW %CVW_SPS %VBOASG %P 2:A2173 = AUS, 3: BOASG
         $OUT[2173] = FALSE
      ;ENDFOLD
      ;FOLD A2174 = EIN ;%{SE}%MKUKATPVW %CVW_SPS %VBOASG %P 2:A2174 = EIN, 3: BOASG
         $OUT[2174] = TRUE
      ;ENDFOLD
      ;FOLD -- Zeit Endlage entprellen -- ;%{SE}%MKUKATPVW %CVW_COM %VCOMMENT %P 2:-- Zeit Endlage entprellen --, 3: VW_COMMENT
      ;ENDFOLD
      ;FOLD t9 ( !E2172 ) = -10[1/10Sek] ;%{SE}%MKUKATPVW %CVW_SPS %VTASG %P 2:t9 ( !E2172 ) = -10[1/10Sek], 3: TASG
         VW(#SET_TIME,NOT $IN[2172],9,0,-10)
      ;ENDFOLD
      ;FOLD Schritt 172 = E2172 & !E2171 & A4039 & T9 + T8  ;%{SE}%MKUKATPVW %CVW_SPS %VST_CON %P 2:Schritt 172 = E2172 & !E2171 & A4039 & T9 + T8 , 3: ST_CON
         IF $IN[2172] AND NOT $IN[2171] AND $OUT[4039] AND $TIMER_FLAG[9] OR $TIMER_FLAG[8] THEN
            PREVSTEP = $APP_INT[5]
            $APP_INT[5] = 172
         ENDIF
      ;ENDFOLD
   ;ENDFOLD
   ;FOLD SCHRITT 172 --MS2 Reinigung (an Pneum. Schwenkeinheit MS2)-- ;%{P}%MKUKATPVW,%CSTEP,%VST_NR,%P 1:SCHRITT, 2:172, 3:MS2 Reinigung (an Pneum. Schwenkeinheit MS2)
      ;FOLD ;%{H}
         Case 172
      ;ENDFOLD
      ;FOLD -- Steuerluft EIN -- ;%{SE}%MKUKATPVW %CVW_COM %VCOMMENT %P 2:-- Steuerluft EIN --, 3: VW_COMMENT
      ;ENDFOLD
      ;FOLD A2169 = A4039 ;%{SE}%MKUKATPVW %CVW_SPS %VBOASG %P 2:A2169 = A4039, 3: BOASG
         $OUT[2169] = $OUT[4039]
      ;ENDFOLD
      ;FOLD -- RSK Fehlerausgabe Schwenkeinheit 2 Arbeitsstellung -- ;%{SE}%MKUKATPVW %CVW_COM %VCOMMENT %P 2:-- RSK Fehlerausgabe Schwenkeinheit 2 Arbeitsstellung --, 3: VW_COMMENT
      ;ENDFOLD
      ;FOLD F324 = !E2172 & T8 + F324 ;%{SE}%MKUKATPVW %CVW_SPS %VBOASG %P 2:F324 = !E2172 & T8 + F324, 3: BOASG
         $FLAG[324] = NOT $IN[2172] AND $TIMER_FLAG[8] OR $FLAG[324]
      ;ENDFOLD
      ;FOLD -- RSK Sammelstoerung -- ;%{SE}%MKUKATPVW %CVW_COM %VCOMMENT %P 2:-- RSK Sammelstoerung --, 3: VW_COMMENT
      ;ENDFOLD
      ;FOLD F329 = F324 ;%{SE}%MKUKATPVW %CVW_SPS %VBOASG %P 2:F329 = F324, 3: BOASG
         $FLAG[329] = $FLAG[324]
      ;ENDFOLD
      ;FOLD A2172 = AUS ;%{SE}%MKUKATPVW %CVW_SPS %VBOASG %P 2:A2172 = AUS, 3: BOASG
         $OUT[2172] = FALSE
      ;ENDFOLD
      ;FOLD -- FRG Bewegung AUS -- ;%{SE}%MKUKATPVW %CVW_COM %VCOMMENT %P 2:-- FRG Bewegung AUS --, 3: VW_COMMENT
      ;ENDFOLD
      ;FOLD A2174 = AUS ;%{SE}%MKUKATPVW %CVW_SPS %VBOASG %P 2:A2174 = AUS, 3: BOASG
         $OUT[2174] = FALSE
      ;ENDFOLD
      ;FOLD -- FRG in Endlage halten ein -- ;%{SE}%MKUKATPVW %CVW_COM %VCOMMENT %P 2:-- FRG in Endlage halten ein --, 3: VW_COMMENT
      ;ENDFOLD
      ;FOLD A2173 = EIN ;%{SE}%MKUKATPVW %CVW_SPS %VBOASG %P 2:A2173 = EIN, 3: BOASG
         $OUT[2173] = TRUE
      ;ENDFOLD
      ;FOLD Schritt 169 = F324 & (E26 + E27) & A4039  ;%{SE}%MKUKATPVW %CVW_SPS %VST_CON %P 2:Schritt 169 = F324 & (E26 + E27) & A4039 , 3: ST_CON
         IF $FLAG[324] AND ($IN[26] OR $IN[27]) AND $OUT[4039] THEN
            PREVSTEP = $APP_INT[5]
            $APP_INT[5] = 169
         ENDIF
      ;ENDFOLD
      ;FOLD Schritt 173 = !F324 & E2172 & A4039  ;%{SE}%MKUKATPVW %CVW_SPS %VST_CON %P 2:Schritt 173 = !F324 & E2172 & A4039 , 3: ST_CON
         IF NOT $FLAG[324] AND $IN[2172] AND $OUT[4039] THEN
            PREVSTEP = $APP_INT[5]
            $APP_INT[5] = 173
         ENDIF
      ;ENDFOLD
   ;ENDFOLD
   ;FOLD SCHRITT 173 --MS2 Reinigung (an Pneum. Schwenkeinheit MS2)-- ;%{P}%MKUKATPVW,%CSTEP,%VST_NR,%P 1:SCHRITT, 2:173, 3:MS2 Reinigung (an Pneum. Schwenkeinheit MS2)
      ;FOLD ;%{H}
         Case 173
      ;ENDFOLD
      ;FOLD -- Steuerluft EIN -- ;%{SE}%MKUKATPVW %CVW_COM %VCOMMENT %P 2:-- Steuerluft EIN --, 3: VW_COMMENT
      ;ENDFOLD
      ;FOLD A2169 = A4039 ;%{SE}%MKUKATPVW %CVW_SPS %VBOASG %P 2:A2169 = A4039, 3: BOASG
         $OUT[2169] = $OUT[4039]
      ;ENDFOLD
      ;FOLD A1896 = AUS ;%{SE}%MKUKATPVW %CVW_SPS %VBOASG %P 2:A1896 = AUS, 3: BOASG
         $OUT[1896] = FALSE
      ;ENDFOLD
      ;FOLD A2175 = AUS ;%{SE}%MKUKATPVW %CVW_SPS %VBOASG %P 2:A2175 = AUS, 3: BOASG
         $OUT[2175] = FALSE
      ;ENDFOLD
      ;FOLD -- Ueberwachungszeit Versetzeinheit -- ;%{SE}%MKUKATPVW %CVW_COM %VCOMMENT %P 2:-- Ueberwachungszeit Versetzeinheit --, 3: VW_COMMENT
      ;ENDFOLD
      ;FOLD t8 ( EIN ) = -100[1/10Sek] ;%{SE}%MKUKATPVW %CVW_SPS %VTASG %P 2:t8 ( EIN ) = -100[1/10Sek], 3: TASG
         VW(#SET_TIME,TRUE,8,0,-100)
      ;ENDFOLD
      ;FOLD Schritt 174 = A4039  ;%{SE}%MKUKATPVW %CVW_SPS %VST_CON %P 2:Schritt 174 = A4039 , 3: ST_CON
         IF $OUT[4039] THEN
            PREVSTEP = $APP_INT[5]
            $APP_INT[5] = 174
         ENDIF
      ;ENDFOLD
   ;ENDFOLD
   ;FOLD SCHRITT 174 --MS2 Reinigung (an Pneum. Schwenkeinheit MS2)-- ;%{P}%MKUKATPVW,%CSTEP,%VST_NR,%P 1:SCHRITT, 2:174, 3:MS2 Reinigung (an Pneum. Schwenkeinheit MS2)
      ;FOLD ;%{H}
         Case 174
      ;ENDFOLD
      ;FOLD -- Steuerluft EIN -- ;%{SE}%MKUKATPVW %CVW_COM %VCOMMENT %P 2:-- Steuerluft EIN --, 3: VW_COMMENT
      ;ENDFOLD
      ;FOLD A2169 = A4039 ;%{SE}%MKUKATPVW %CVW_SPS %VBOASG %P 2:A2169 = A4039, 3: BOASG
         $OUT[2169] = $OUT[4039]
      ;ENDFOLD
      ;FOLD -- RSK Fehlerausgabe Versetzeinheit -- ;%{SE}%MKUKATPVW %CVW_COM %VCOMMENT %P 2:-- RSK Fehlerausgabe Versetzeinheit --, 3: VW_COMMENT
      ;ENDFOLD
      ;FOLD F328 = F585 & T8 ;%{SE}%MKUKATPVW %CVW_SPS %VBOASG %P 2:F328 = F585 & T8, 3: BOASG
         $FLAG[328] = $FLAG[585] AND $TIMER_FLAG[8]
      ;ENDFOLD
      ;FOLD -- RSK Sammelstoerung -- ;%{SE}%MKUKATPVW %CVW_COM %VCOMMENT %P 2:-- RSK Sammelstoerung --, 3: VW_COMMENT
      ;ENDFOLD
      ;FOLD F329 = T8 ;%{SE}%MKUKATPVW %CVW_SPS %VBOASG %P 2:F329 = T8, 3: BOASG
         $FLAG[329] = $TIMER_FLAG[8]
      ;ENDFOLD
      ;FOLD -- Versetzeinheit in Arbeitsst. schw. -- ;%{SE}%MKUKATPVW %CVW_COM %VCOMMENT %P 2:-- Versetzeinheit in Arbeitsst. schw. --, 3: VW_COMMENT
      ;ENDFOLD
      ;FOLD A2176 = !E2176 & E2172 & F585 ;%{SE}%MKUKATPVW %CVW_SPS %VBOASG %P 2:A2176 = !E2176 & E2172 & F585, 3: BOASG
         $OUT[2176] = NOT $IN[2176] AND $IN[2172] AND $FLAG[585]
      ;ENDFOLD
      ;FOLD Schritt 173 = A2176 & T8 & (E26 + E27) & A4039  ;%{SE}%MKUKATPVW %CVW_SPS %VST_CON %P 2:Schritt 173 = A2176 & T8 & (E26 + E27) & A4039 , 3: ST_CON
         IF $OUT[2176] AND $TIMER_FLAG[8] AND ($IN[26] OR $IN[27]) AND $OUT[4039] THEN
            PREVSTEP = $APP_INT[5]
            $APP_INT[5] = 173
         ENDIF
      ;ENDFOLD
      ;FOLD Schritt 175 = (E2176 & F585 + !E2168 & !F585) & A4039  ;%{SE}%MKUKATPVW %CVW_SPS %VST_CON %P 2:Schritt 175 = (E2176 & F585 + !E2168 & !F585) & A4039 , 3: ST_CON
         IF ($IN[2176] AND $FLAG[585] OR NOT $IN[2168] AND NOT $FLAG[585]) AND $OUT[4039] THEN
            PREVSTEP = $APP_INT[5]
            $APP_INT[5] = 175
         ENDIF
      ;ENDFOLD
   ;ENDFOLD
   ;FOLD SCHRITT 175 --MS2 Reinigung (an Pneum.  Schwenkeinheit  MS2)-- ;%{P}%MKUKATPVW,%CSTEP,%VST_NR,%P 1:SCHRITT, 2:175, 3:MS2 Reinigung (an Pneum.  Schwenkeinheit  MS2)
      ;FOLD ;%{H}
         Case 175
      ;ENDFOLD
      ;FOLD -- Steuerluft EIN -- ;%{SE}%MKUKATPVW %CVW_COM %VCOMMENT %P 2:-- Steuerluft EIN --, 3: VW_COMMENT
      ;ENDFOLD
      ;FOLD A2169 = A4039 ;%{SE}%MKUKATPVW %CVW_SPS %VBOASG %P 2:A2169 = A4039, 3: BOASG
         $OUT[2169] = $OUT[4039]
      ;ENDFOLD
      ;FOLD -- RSK Sammelstoerung -- ;%{SE}%MKUKATPVW %CVW_COM %VCOMMENT %P 2:-- RSK Sammelstoerung --, 3: VW_COMMENT
      ;ENDFOLD
      ;FOLD F329 = T8 ;%{SE}%MKUKATPVW %CVW_SPS %VBOASG %P 2:F329 = T8, 3: BOASG
         $FLAG[329] = $TIMER_FLAG[8]
      ;ENDFOLD
      ;FOLD -- Zeit Reinigung -- ;%{SE}%MKUKATPVW %CVW_COM %VCOMMENT %P 2:-- Zeit Reinigung --, 3: VW_COMMENT
      ;ENDFOLD
      ;FOLD F271 = i26 = 0 ;%{SE}%MKUKATPVW %CVW_SPS %VBOCMP %P 2:F271 = i26 = 0, 3: BOCMP
         $FLAG[271] = $COUNT_I[26] == 0
      ;ENDFOLD
      ;FOLD t9 ( F271 ) = -20[1/10Sek] ;%{SE}%MKUKATPVW %CVW_SPS %VTASG %P 2:t9 ( F271 ) = -20[1/10Sek], 3: TASG
         VW(#SET_TIME,$FLAG[271],9,0,-20)
      ;ENDFOLD
      ;FOLD t9 ( !F271 ) = i26[1/10Sek] ;%{SE}%MKUKATPVW %CVW_SPS %VTASG %P 2:t9 ( !F271 ) = i26[1/10Sek], 3: TASG
         VW(#SET_TIME,NOT $FLAG[271],9,0,$COUNT_I[26])
      ;ENDFOLD
      ;FOLD -- MS2 Ausblasen EIN -- ;%{SE}%MKUKATPVW %CVW_COM %VCOMMENT %P 2:-- MS2 Ausblasen EIN --, 3: VW_COMMENT
      ;ENDFOLD
      ;FOLD A1902 = EIN ;%{SE}%MKUKATPVW %CVW_SPS %VBOASG %P 2:A1902 = EIN, 3: BOASG
         $OUT[1902] = TRUE
      ;ENDFOLD
      ;FOLD -- MS2 Reinigung starten -- ;%{SE}%MKUKATPVW %CVW_COM %VCOMMENT %P 2:-- MS2 Reinigung starten --, 3: VW_COMMENT
      ;ENDFOLD
      ;FOLD A1896 = EIN ;%{SE}%MKUKATPVW %CVW_SPS %VBOASG %P 2:A1896 = EIN, 3: BOASG
         $OUT[1896] = TRUE
      ;ENDFOLD
      ;FOLD Schritt 173 = E1896 & T8 & (E26 + E27) & A4039  ;%{SE}%MKUKATPVW %CVW_SPS %VST_CON %P 2:Schritt 173 = E1896 & T8 & (E26 + E27) & A4039 , 3: ST_CON
         IF $IN[1896] AND $TIMER_FLAG[8] AND ($IN[26] OR $IN[27]) AND $OUT[4039] THEN
            PREVSTEP = $APP_INT[5]
            $APP_INT[5] = 173
         ENDIF
      ;ENDFOLD
      ;FOLD Schritt 176 = !E1896 & A4039  ;%{SE}%MKUKATPVW %CVW_SPS %VST_CON %P 2:Schritt 176 = !E1896 & A4039 , 3: ST_CON
         IF NOT $IN[1896] AND $OUT[4039] THEN
            PREVSTEP = $APP_INT[5]
            $APP_INT[5] = 176
         ENDIF
      ;ENDFOLD
   ;ENDFOLD
   ;FOLD SCHRITT 176 --MS2 Reinigung (an Pneum.  Schwenkeinheit  MS2)-- ;%{P}%MKUKATPVW,%CSTEP,%VST_NR,%P 1:SCHRITT, 2:176, 3:MS2 Reinigung (an Pneum.  Schwenkeinheit  MS2)
      ;FOLD ;%{H}
         Case 176
      ;ENDFOLD
      ;FOLD -- Steuerluft EIN -- ;%{SE}%MKUKATPVW %CVW_COM %VCOMMENT %P 2:-- Steuerluft EIN --, 3: VW_COMMENT
      ;ENDFOLD
      ;FOLD A2169 = A4039 ;%{SE}%MKUKATPVW %CVW_SPS %VBOASG %P 2:A2169 = A4039, 3: BOASG
         $OUT[2169] = $OUT[4039]
      ;ENDFOLD
      ;FOLD Schritt 173 = !E1896 & T9 & (E26 + E27) & A4039  ;%{SE}%MKUKATPVW %CVW_SPS %VST_CON %P 2:Schritt 173 = !E1896 & T9 & (E26 + E27) & A4039 , 3: ST_CON
         IF NOT $IN[1896] AND $TIMER_FLAG[9] AND ($IN[26] OR $IN[27]) AND $OUT[4039] THEN
            PREVSTEP = $APP_INT[5]
            $APP_INT[5] = 173
         ENDIF
      ;ENDFOLD
      ;FOLD Schritt 177 = T9 & A4039  ;%{SE}%MKUKATPVW %CVW_SPS %VST_CON %P 2:Schritt 177 = T9 & A4039 , 3: ST_CON
         IF $TIMER_FLAG[9] AND $OUT[4039] THEN
            PREVSTEP = $APP_INT[5]
            $APP_INT[5] = 177
         ENDIF
      ;ENDFOLD
   ;ENDFOLD
   ;FOLD SCHRITT 177 --MS2 Reinigung (an Pneum. Schwenkeinheit MS2)-- ;%{P}%MKUKATPVW,%CSTEP,%VST_NR,%P 1:SCHRITT, 2:177, 3:MS2 Reinigung (an Pneum. Schwenkeinheit MS2)
      ;FOLD ;%{H}
         Case 177
      ;ENDFOLD
      ;FOLD -- Steuerluft EIN -- ;%{SE}%MKUKATPVW %CVW_COM %VCOMMENT %P 2:-- Steuerluft EIN --, 3: VW_COMMENT
      ;ENDFOLD
      ;FOLD A2169 = A4039 ;%{SE}%MKUKATPVW %CVW_SPS %VBOASG %P 2:A2169 = A4039, 3: BOASG
         $OUT[2169] = $OUT[4039]
      ;ENDFOLD
      ;FOLD -- RSK Sammelstoerung -- ;%{SE}%MKUKATPVW %CVW_COM %VCOMMENT %P 2:-- RSK Sammelstoerung --, 3: VW_COMMENT
      ;ENDFOLD
      ;FOLD F329 = T8 ;%{SE}%MKUKATPVW %CVW_SPS %VBOASG %P 2:F329 = T8, 3: BOASG
         $FLAG[329] = $TIMER_FLAG[8]
      ;ENDFOLD
      ;FOLD -- MS2 Reinigung beenden -- ;%{SE}%MKUKATPVW %CVW_COM %VCOMMENT %P 2:-- MS2 Reinigung beenden --, 3: VW_COMMENT
      ;ENDFOLD
      ;FOLD A1896 = AUS ;%{SE}%MKUKATPVW %CVW_SPS %VBOASG %P 2:A1896 = AUS, 3: BOASG
         $OUT[1896] = FALSE
      ;ENDFOLD
      ;FOLD -- MS2 Ausblasen AUS -- ;%{SE}%MKUKATPVW %CVW_COM %VCOMMENT %P 2:-- MS2 Ausblasen AUS --, 3: VW_COMMENT
      ;ENDFOLD
      ;FOLD A1902 = AUS ;%{SE}%MKUKATPVW %CVW_SPS %VBOASG %P 2:A1902 = AUS, 3: BOASG
         $OUT[1902] = FALSE
      ;ENDFOLD
      ;FOLD -- MS2 Einspruehen EIN -- ;%{SE}%MKUKATPVW %CVW_COM %VCOMMENT %P 2:-- MS2 Einspruehen EIN --, 3: VW_COMMENT
      ;ENDFOLD
      ;FOLD A528 = !F583 & F584 ;%{SE}%MKUKATPVW %CVW_SPS %VBOASG %P 2:A528 = !F583 & F584, 3: BOASG
         $OUT[528] = NOT $FLAG[583] AND $FLAG[584]
      ;ENDFOLD
      ;FOLD A1903 = F583 & F584 ;%{SE}%MKUKATPVW %CVW_SPS %VBOASG %P 2:A1903 = F583 & F584, 3: BOASG
         $OUT[1903] = $FLAG[583] AND $FLAG[584]
      ;ENDFOLD
      ;FOLD -- Einschaltdauer Einspruehen -- ;%{SE}%MKUKATPVW %CVW_COM %VCOMMENT %P 2:-- Einschaltdauer Einspruehen --, 3: VW_COMMENT
      ;ENDFOLD
      ;FOLD t7 ( EIN ) = i23[1/10Sek] ;%{SE}%MKUKATPVW %CVW_SPS %VTASG %P 2:t7 ( EIN ) = i23[1/10Sek], 3: TASG
         VW(#SET_TIME,TRUE,7,0,$COUNT_I[23])
      ;ENDFOLD
      ;FOLD Schritt 178 = A4039  ;%{SE}%MKUKATPVW %CVW_SPS %VST_CON %P 2:Schritt 178 = A4039 , 3: ST_CON
         IF $OUT[4039] THEN
            PREVSTEP = $APP_INT[5]
            $APP_INT[5] = 178
         ENDIF
      ;ENDFOLD
   ;ENDFOLD
   ;FOLD SCHRITT 178 --MS2 Reinigung (an Pneum. Schwenkeinheit MS2)-- ;%{P}%MKUKATPVW,%CSTEP,%VST_NR,%P 1:SCHRITT, 2:178, 3:MS2 Reinigung (an Pneum. Schwenkeinheit MS2)
      ;FOLD ;%{H}
         Case 178
      ;ENDFOLD
      ;FOLD F323 = AUS ;%{SE}%MKUKATPVW %CVW_SPS %VBOASG %P 2:F323 = AUS, 3: BOASG
         $FLAG[323] = FALSE
      ;ENDFOLD
      ;FOLD A2171 = AUS ;%{SE}%MKUKATPVW %CVW_SPS %VBOASG %P 2:A2171 = AUS, 3: BOASG
         $OUT[2171] = FALSE
      ;ENDFOLD
      ;FOLD A2172 = AUS ;%{SE}%MKUKATPVW %CVW_SPS %VBOASG %P 2:A2172 = AUS, 3: BOASG
         $OUT[2172] = FALSE
      ;ENDFOLD
      ;FOLD A2173 = AUS ;%{SE}%MKUKATPVW %CVW_SPS %VBOASG %P 2:A2173 = AUS, 3: BOASG
         $OUT[2173] = FALSE
      ;ENDFOLD
      ;FOLD A2174 = AUS ;%{SE}%MKUKATPVW %CVW_SPS %VBOASG %P 2:A2174 = AUS, 3: BOASG
         $OUT[2174] = FALSE
      ;ENDFOLD
      ;FOLD A2175 = AUS ;%{SE}%MKUKATPVW %CVW_SPS %VBOASG %P 2:A2175 = AUS, 3: BOASG
         $OUT[2175] = FALSE
      ;ENDFOLD
      ;FOLD -- Ueberwachungszeit Schwenkeinheit 2 schwenken -- ;%{SE}%MKUKATPVW %CVW_COM %VCOMMENT %P 2:-- Ueberwachungszeit Schwenkeinheit 2 schwenken --, 3: VW_COMMENT
      ;ENDFOLD
      ;FOLD t8 ( EIN ) = -100[1/10Sek] ;%{SE}%MKUKATPVW %CVW_SPS %VTASG %P 2:t8 ( EIN ) = -100[1/10Sek], 3: TASG
         VW(#SET_TIME,TRUE,8,0,-100)
      ;ENDFOLD
      ;FOLD Schritt 179 = T7 & A4039  ;%{SE}%MKUKATPVW %CVW_SPS %VST_CON %P 2:Schritt 179 = T7 & A4039 , 3: ST_CON
         IF $TIMER_FLAG[7] AND $OUT[4039] THEN
            PREVSTEP = $APP_INT[5]
            $APP_INT[5] = 179
         ENDIF
      ;ENDFOLD
   ;ENDFOLD
   ;FOLD SCHRITT 179 --MS2 Reinigung (an Pneum. Schwenkeinheit MS2)-- ;%{P}%MKUKATPVW,%CSTEP,%VST_NR,%P 1:SCHRITT, 2:179, 3:MS2 Reinigung (an Pneum. Schwenkeinheit MS2)
      ;FOLD ;%{H}
         Case 179
      ;ENDFOLD
      ;FOLD -- Steuerluft EIN -- ;%{SE}%MKUKATPVW %CVW_COM %VCOMMENT %P 2:-- Steuerluft EIN --, 3: VW_COMMENT
      ;ENDFOLD
      ;FOLD A2169 = A4039 ;%{SE}%MKUKATPVW %CVW_SPS %VBOASG %P 2:A2169 = A4039, 3: BOASG
         $OUT[2169] = $OUT[4039]
      ;ENDFOLD
      ;FOLD -- MS2 Einspruehen AUS -- ;%{SE}%MKUKATPVW %CVW_COM %VCOMMENT %P 2:-- MS2 Einspruehen AUS --, 3: VW_COMMENT
      ;ENDFOLD
      ;FOLD A528 = AUS ;%{SE}%MKUKATPVW %CVW_SPS %VBOASG %P 2:A528 = AUS, 3: BOASG
         $OUT[528] = FALSE
      ;ENDFOLD
      ;FOLD A1903 = AUS ;%{SE}%MKUKATPVW %CVW_SPS %VBOASG %P 2:A1903 = AUS, 3: BOASG
         $OUT[1903] = FALSE
      ;ENDFOLD
      ;FOLD -- Versetzeinheit in Ruhest. schw. -- ;%{SE}%MKUKATPVW %CVW_COM %VCOMMENT %P 2:-- Versetzeinheit in Ruhest. schw. --, 3: VW_COMMENT
      ;ENDFOLD
      ;FOLD A2175 = EIN ;%{SE}%MKUKATPVW %CVW_SPS %VBOASG %P 2:A2175 = EIN, 3: BOASG
         $OUT[2175] = TRUE
      ;ENDFOLD
      ;FOLD A2176 = AUS ;%{SE}%MKUKATPVW %CVW_SPS %VBOASG %P 2:A2176 = AUS, 3: BOASG
         $OUT[2176] = FALSE
      ;ENDFOLD
      ;FOLD -- RSK Fehlerausgabe Versetzeinheit in Ruhest. schw. -- ;%{SE}%MKUKATPVW %CVW_COM %VCOMMENT %P 2:-- RSK Fehlerausgabe Versetzeinheit in Ruhest. schw. --, 3: VW_COMMENT
      ;ENDFOLD
      ;FOLD F328 = F585 & T8 ;%{SE}%MKUKATPVW %CVW_SPS %VBOASG %P 2:F328 = F585 & T8, 3: BOASG
         $FLAG[328] = $FLAG[585] AND $TIMER_FLAG[8]
      ;ENDFOLD
      ;FOLD -- RSK Fehlerausgabe Schwenkeinheit 2 Arbeit. -- ;%{SE}%MKUKATPVW %CVW_COM %VCOMMENT %P 2:-- RSK Fehlerausgabe Schwenkeinheit 2 Arbeit. --, 3: VW_COMMENT
      ;ENDFOLD
      ;FOLD F324 = !E2172 & T8 ;%{SE}%MKUKATPVW %CVW_SPS %VBOASG %P 2:F324 = !E2172 & T8, 3: BOASG
         $FLAG[324] = NOT $IN[2172] AND $TIMER_FLAG[8]
      ;ENDFOLD
      ;FOLD -- RSK Sammelstoerung -- ;%{SE}%MKUKATPVW %CVW_COM %VCOMMENT %P 2:-- RSK Sammelstoerung --, 3: VW_COMMENT
      ;ENDFOLD
      ;FOLD F329 = F324 + F328 ;%{SE}%MKUKATPVW %CVW_SPS %VBOASG %P 2:F329 = F324 + F328, 3: BOASG
         $FLAG[329] = $FLAG[324] OR $FLAG[328]
      ;ENDFOLD
      ;FOLD Schritt 178 = (E26 + E27) & (F324 + F328) & A4039  ;%{SE}%MKUKATPVW %CVW_SPS %VST_CON %P 2:Schritt 178 = (E26 + E27) & (F324 + F328) & A4039 , 3: ST_CON
         IF ($IN[26] OR $IN[27]) AND ($FLAG[324] OR $FLAG[328]) AND $OUT[4039] THEN
            PREVSTEP = $APP_INT[5]
            $APP_INT[5] = 178
         ENDIF
      ;ENDFOLD
      ;FOLD Schritt 180 = (!F324 + T8) & (F523 & !F524 & E2169 + !F523 & F524 & !E2170) & E2175 & F585 & A4039  ;%{SE}%MKUKATPVW %CVW_SPS %VST_CON %P 2:Schritt 180 = (!F324 + T8) & (F523 & !F524 & E2169 + !F523 & F524 & !E2170) & E2175 & F585 & A4039 , 3: ST_CON
         IF (NOT $FLAG[324] OR $TIMER_FLAG[8]) AND ($FLAG[523] AND NOT $FLAG[524] AND $IN[2169] OR NOT $FLAG[523] AND $FLAG[524] AND NOT $IN[2170]) AND $IN[2175] AND $FLAG[585] AND $OUT[4039] THEN
            PREVSTEP = $APP_INT[5]
            $APP_INT[5] = 180
         ENDIF
      ;ENDFOLD
      ;FOLD Schritt 180 = (!F324 + T8) & (F523 & !F524 & E2169 + !F523 & F524 & !E2170) & !E2175 & !F585 & A4039  ;%{SE}%MKUKATPVW %CVW_SPS %VST_CON %P 2:Schritt 180 = (!F324 + T8) & (F523 & !F524 & E2169 + !F523 & F524 & !E2170) & !E2175 & !F585 & A4039 , 3: ST_CON
         IF (NOT $FLAG[324] OR $TIMER_FLAG[8]) AND ($FLAG[523] AND NOT $FLAG[524] AND $IN[2169] OR NOT $FLAG[523] AND $FLAG[524] AND NOT $IN[2170]) AND NOT $IN[2175] AND NOT $FLAG[585] AND $OUT[4039] THEN
            PREVSTEP = $APP_INT[5]
            $APP_INT[5] = 180
         ENDIF
      ;ENDFOLD
   ;ENDFOLD
   ;FOLD SCHRITT 180 --MS2 Reinigung (an Pneum. Schwenkeinheit MS2)-- ;%{P}%MKUKATPVW,%CSTEP,%VST_NR,%P 1:SCHRITT, 2:180, 3:MS2 Reinigung (an Pneum. Schwenkeinheit MS2)
      ;FOLD ;%{H}
         Case 180
      ;ENDFOLD
      ;FOLD -- Steuerluft EIN -- ;%{SE}%MKUKATPVW %CVW_COM %VCOMMENT %P 2:-- Steuerluft EIN --, 3: VW_COMMENT
      ;ENDFOLD
      ;FOLD A2169 = A4039 ;%{SE}%MKUKATPVW %CVW_SPS %VBOASG %P 2:A2169 = A4039, 3: BOASG
         $OUT[2169] = $OUT[4039]
      ;ENDFOLD
      ;FOLD A2176 = AUS ;%{SE}%MKUKATPVW %CVW_SPS %VBOASG %P 2:A2176 = AUS, 3: BOASG
         $OUT[2176] = FALSE
      ;ENDFOLD
      ;FOLD -- Schwenkeinheit 2 in Ruhestellung schwenken -- ;%{SE}%MKUKATPVW %CVW_COM %VCOMMENT %P 2:-- Schwenkeinheit 2 in Ruhestellung schwenken --, 3: VW_COMMENT
      ;ENDFOLD
      ;FOLD A2171 = !E2171 ;%{SE}%MKUKATPVW %CVW_SPS %VBOASG %P 2:A2171 = !E2171, 3: BOASG
         $OUT[2171] = NOT $IN[2171]
      ;ENDFOLD
      ;FOLD A2172 = AUS ;%{SE}%MKUKATPVW %CVW_SPS %VBOASG %P 2:A2172 = AUS, 3: BOASG
         $OUT[2172] = FALSE
      ;ENDFOLD
      ;FOLD -- FRG Bewegung EIN -- ;%{SE}%MKUKATPVW %CVW_COM %VCOMMENT %P 2:-- FRG Bewegung EIN --, 3: VW_COMMENT
      ;ENDFOLD
      ;FOLD A2173 = AUS ;%{SE}%MKUKATPVW %CVW_SPS %VBOASG %P 2:A2173 = AUS, 3: BOASG
         $OUT[2173] = FALSE
      ;ENDFOLD
      ;FOLD A2174 = !E2171 ;%{SE}%MKUKATPVW %CVW_SPS %VBOASG %P 2:A2174 = !E2171, 3: BOASG
         $OUT[2174] = NOT $IN[2171]
      ;ENDFOLD
      ;FOLD Schritt 181 = E1896 & !E2172 & E2171 & A4039  + T8  ;%{SE}%MKUKATPVW %CVW_SPS %VST_CON %P 2:Schritt 181 = E1896 & !E2172 & E2171 & A4039  + T8 , 3: ST_CON
         IF $IN[1896] AND NOT $IN[2172] AND $IN[2171] AND $OUT[4039] OR $TIMER_FLAG[8] THEN
            PREVSTEP = $APP_INT[5]
            $APP_INT[5] = 181
         ENDIF
      ;ENDFOLD
   ;ENDFOLD
   ;FOLD SCHRITT 181 --MS2 Reinigung (an Pneum. Schwenkeinheit MS2)-- ;%{P}%MKUKATPVW,%CSTEP,%VST_NR,%P 1:SCHRITT, 2:181, 3:MS2 Reinigung (an Pneum. Schwenkeinheit MS2)
      ;FOLD ;%{H}
         Case 181
      ;ENDFOLD
      ;FOLD -- Steuerluft EIN -- ;%{SE}%MKUKATPVW %CVW_COM %VCOMMENT %P 2:-- Steuerluft EIN --, 3: VW_COMMENT
      ;ENDFOLD
      ;FOLD A2169 = A4039 ;%{SE}%MKUKATPVW %CVW_SPS %VBOASG %P 2:A2169 = A4039, 3: BOASG
         $OUT[2169] = $OUT[4039]
      ;ENDFOLD
      ;FOLD -- RSK Fehlerausgabe Schwenkeinheit 2 Ruhestellung -- ;%{SE}%MKUKATPVW %CVW_COM %VCOMMENT %P 2:-- RSK Fehlerausgabe Schwenkeinheit 2 Ruhestellung --, 3: VW_COMMENT
      ;ENDFOLD
      ;FOLD F323 = !E2171 & T8 + F323 ;%{SE}%MKUKATPVW %CVW_SPS %VBOASG %P 2:F323 = !E2171 & T8 + F323, 3: BOASG
         $FLAG[323] = NOT $IN[2171] AND $TIMER_FLAG[8] OR $FLAG[323]
      ;ENDFOLD
      ;FOLD -- RSK Sammelstoerung -- ;%{SE}%MKUKATPVW %CVW_COM %VCOMMENT %P 2:-- RSK Sammelstoerung --, 3: VW_COMMENT
      ;ENDFOLD
      ;FOLD F329 = F323 ;%{SE}%MKUKATPVW %CVW_SPS %VBOASG %P 2:F329 = F323, 3: BOASG
         $FLAG[329] = $FLAG[323]
      ;ENDFOLD
      ;FOLD A2171 = AUS ;%{SE}%MKUKATPVW %CVW_SPS %VBOASG %P 2:A2171 = AUS, 3: BOASG
         $OUT[2171] = FALSE
      ;ENDFOLD
      ;FOLD -- FRG Bewegung AUS -- ;%{SE}%MKUKATPVW %CVW_COM %VCOMMENT %P 2:-- FRG Bewegung AUS --, 3: VW_COMMENT
      ;ENDFOLD
      ;FOLD A2174 = AUS ;%{SE}%MKUKATPVW %CVW_SPS %VBOASG %P 2:A2174 = AUS, 3: BOASG
         $OUT[2174] = FALSE
      ;ENDFOLD
      ;FOLD Schritt 178 = F323 & (E26 + E27) & A4039  ;%{SE}%MKUKATPVW %CVW_SPS %VST_CON %P 2:Schritt 178 = F323 & (E26 + E27) & A4039 , 3: ST_CON
         IF $FLAG[323] AND ($IN[26] OR $IN[27]) AND $OUT[4039] THEN
            PREVSTEP = $APP_INT[5]
            $APP_INT[5] = 178
         ENDIF
      ;ENDFOLD
      ;FOLD Schritt 182 = !F323 & (E2174 + F837) & A4039  ;%{SE}%MKUKATPVW %CVW_SPS %VST_CON %P 2:Schritt 182 = !F323 & (E2174 + F837) & A4039 , 3: ST_CON
         IF NOT $FLAG[323] AND ($IN[2174] OR $FLAG[837]) AND $OUT[4039] THEN
            PREVSTEP = $APP_INT[5]
            $APP_INT[5] = 182
         ENDIF
      ;ENDFOLD
   ;ENDFOLD
   ;FOLD SCHRITT 182 --MS2 Reinigung (an Pneum. Schwenkeinheit MS2)-- ;%{P}%MKUKATPVW,%CSTEP,%VST_NR,%P 1:SCHRITT, 2:182, 3:MS2 Reinigung (an Pneum. Schwenkeinheit MS2)
      ;FOLD ;%{H}
         Case 182
      ;ENDFOLD
      ;FOLD -- Steuerluft EIN -- ;%{SE}%MKUKATPVW %CVW_COM %VCOMMENT %P 2:-- Steuerluft EIN --, 3: VW_COMMENT
      ;ENDFOLD
      ;FOLD A2169 = A4039 ;%{SE}%MKUKATPVW %CVW_SPS %VBOASG %P 2:A2169 = A4039, 3: BOASG
         $OUT[2169] = $OUT[4039]
      ;ENDFOLD
      ;FOLD F329 = T8 ;%{SE}%MKUKATPVW %CVW_SPS %VBOASG %P 2:F329 = T8, 3: BOASG
         $FLAG[329] = $TIMER_FLAG[8]
      ;ENDFOLD
      ;FOLD F323 = AUS ;%{SE}%MKUKATPVW %CVW_SPS %VBOASG %P 2:F323 = AUS, 3: BOASG
         $FLAG[323] = FALSE
      ;ENDFOLD
      ;FOLD -- FRG in Endlage halten ein -- ;%{SE}%MKUKATPVW %CVW_COM %VCOMMENT %P 2:-- FRG in Endlage halten ein --, 3: VW_COMMENT
      ;ENDFOLD
      ;FOLD A2173 = EIN ;%{SE}%MKUKATPVW %CVW_SPS %VBOASG %P 2:A2173 = EIN, 3: BOASG
         $OUT[2173] = TRUE
      ;ENDFOLD
      ;FOLD Schritt 183 = !E2173 & (E2174 + F837) & A4039  ;%{SE}%MKUKATPVW %CVW_SPS %VST_CON %P 2:Schritt 183 = !E2173 & (E2174 + F837) & A4039 , 3: ST_CON
         IF NOT $IN[2173] AND ($IN[2174] OR $FLAG[837]) AND $OUT[4039] THEN
            PREVSTEP = $APP_INT[5]
            $APP_INT[5] = 183
         ENDIF
      ;ENDFOLD
   ;ENDFOLD
   ;FOLD SCHRITT 183 --MS2 Reinigung (an Pneum. Schwenkeinheit MS2)-- ;%{P}%MKUKATPVW,%CSTEP,%VST_NR,%P 1:SCHRITT, 2:183, 3:MS2 Reinigung (an Pneum. Schwenkeinheit MS2)
      ;FOLD ;%{H}
         Case 183
      ;ENDFOLD
      ;FOLD -- Steuerluft EIN -- ;%{SE}%MKUKATPVW %CVW_COM %VCOMMENT %P 2:-- Steuerluft EIN --, 3: VW_COMMENT
      ;ENDFOLD
      ;FOLD A2169 = A4039 ;%{SE}%MKUKATPVW %CVW_SPS %VBOASG %P 2:A2169 = A4039, 3: BOASG
         $OUT[2169] = $OUT[4039]
      ;ENDFOLD
      ;FOLD -- FRG in Endlage halten AUS -- ;%{SE}%MKUKATPVW %CVW_COM %VCOMMENT %P 2:-- FRG in Endlage halten AUS --, 3: VW_COMMENT
      ;ENDFOLD
      ;FOLD A2173 = AUS ;%{SE}%MKUKATPVW %CVW_SPS %VBOASG %P 2:A2173 = AUS, 3: BOASG
         $OUT[2173] = FALSE
      ;ENDFOLD
      ;FOLD -- MS1 Zaehler ruecksetzen -- ;%{SE}%MKUKATPVW %CVW_COM %VCOMMENT %P 2:-- MS1 Zaehler ruecksetzen --, 3: VW_COMMENT
      ;ENDFOLD
      ;FOLD -- MS1 FRG Reinigung -- ;%{SE}%MKUKATPVW %CVW_COM %VCOMMENT %P 2:-- MS1 FRG Reinigung --, 3: VW_COMMENT
      ;ENDFOLD
      ;FOLD F607 = AUS ;%{SE}%MKUKATPVW %CVW_SPS %VBOASG %P 2:F607 = AUS, 3: BOASG
         $FLAG[607] = FALSE
      ;ENDFOLD
      ;FOLD -- MS1 Reinigung FK -- ;%{SE}%MKUKATPVW %CVW_COM %VCOMMENT %P 2:-- MS1 Reinigung FK --, 3: VW_COMMENT
      ;ENDFOLD
      ;FOLD F609 = EIN ;%{SE}%MKUKATPVW %CVW_SPS %VBOASG %P 2:F609 = EIN, 3: BOASG
         $FLAG[609] = TRUE
      ;ENDFOLD
      ;FOLD t8 ( EIN ) = STOP ;%{SE}%MKUKATPVW %CVW_SPS %VTSTOP %P 2:t8 ( EIN ) = STOP, 3: TSTOP
         VW(#SET_TIME,TRUE,8,1,0)
      ;ENDFOLD
      ;FOLD Schritt 1 = A4039  ;%{SE}%MKUKATPVW %CVW_SPS %VST_CON %P 2:Schritt 1 = A4039 , 3: ST_CON
         IF $OUT[4039] THEN
            PREVSTEP = $APP_INT[5]
            $APP_INT[5] = 1
         ENDIF
      ;ENDFOLD
   ;ENDFOLD
   ;FOLD SCHRITT 184 --KL1 Spueleimer (an Pneum. Schwenkeinheit KL1)-- ;%{P}%MKUKATPVW,%CSTEP,%VST_NR,%P 1:SCHRITT, 2:184, 3:KL1 Spueleimer (an Pneum. Schwenkeinheit KL1)
      ;FOLD ;%{H}
         Case 184
      ;ENDFOLD
      ;FOLD -- RSK gestartet -- ;%{SE}%MKUKATPVW %CVW_COM %VCOMMENT %P 2:-- RSK gestartet --, 3: VW_COMMENT
      ;ENDFOLD
      ;FOLD F321 = AUS ;%{SE}%MKUKATPVW %CVW_SPS %VBOASG %P 2:F321 = AUS, 3: BOASG
         $FLAG[321] = FALSE
      ;ENDFOLD
      ;FOLD F323 = AUS ;%{SE}%MKUKATPVW %CVW_SPS %VBOASG %P 2:F323 = AUS, 3: BOASG
         $FLAG[323] = FALSE
      ;ENDFOLD
      ;FOLD F324 = AUS ;%{SE}%MKUKATPVW %CVW_SPS %VBOASG %P 2:F324 = AUS, 3: BOASG
         $FLAG[324] = FALSE
      ;ENDFOLD
      ;FOLD F329 = AUS ;%{SE}%MKUKATPVW %CVW_SPS %VBOASG %P 2:F329 = AUS, 3: BOASG
         $FLAG[329] = FALSE
      ;ENDFOLD
      ;FOLD A161 = EIN ;%{SE}%MKUKATPVW %CVW_SPS %VBOASG %P 2:A161 = EIN, 3: BOASG
         $OUT[161] = TRUE
      ;ENDFOLD
      ;FOLD -- Steuerluft EIN -- ;%{SE}%MKUKATPVW %CVW_COM %VCOMMENT %P 2:-- Steuerluft EIN --, 3: VW_COMMENT
      ;ENDFOLD
      ;FOLD A2113 = A4039 ;%{SE}%MKUKATPVW %CVW_SPS %VBOASG %P 2:A2113 = A4039, 3: BOASG
         $OUT[2113] = $OUT[4039]
      ;ENDFOLD
      ;FOLD A2115 = AUS ;%{SE}%MKUKATPVW %CVW_SPS %VBOASG %P 2:A2115 = AUS, 3: BOASG
         $OUT[2115] = FALSE
      ;ENDFOLD
      ;FOLD A2116 = AUS ;%{SE}%MKUKATPVW %CVW_SPS %VBOASG %P 2:A2116 = AUS, 3: BOASG
         $OUT[2116] = FALSE
      ;ENDFOLD
      ;FOLD A2117 = AUS ;%{SE}%MKUKATPVW %CVW_SPS %VBOASG %P 2:A2117 = AUS, 3: BOASG
         $OUT[2117] = FALSE
      ;ENDFOLD
      ;FOLD A2118 = AUS ;%{SE}%MKUKATPVW %CVW_SPS %VBOASG %P 2:A2118 = AUS, 3: BOASG
         $OUT[2118] = FALSE
      ;ENDFOLD
      ;FOLD -- Ueberwachungszeit Schwenkeinheit 1 -- ;%{SE}%MKUKATPVW %CVW_COM %VCOMMENT %P 2:-- Ueberwachungszeit Schwenkeinheit 1 --, 3: VW_COMMENT
      ;ENDFOLD
      ;FOLD t8 ( EIN ) = -100[1/10Sek] ;%{SE}%MKUKATPVW %CVW_SPS %VTASG %P 2:t8 ( EIN ) = -100[1/10Sek], 3: TASG
         VW(#SET_TIME,TRUE,8,0,-100)
      ;ENDFOLD
      ;FOLD Schritt 185 = !E2116 & A4039  ;%{SE}%MKUKATPVW %CVW_SPS %VST_CON %P 2:Schritt 185 = !E2116 & A4039 , 3: ST_CON
         IF NOT $IN[2116] AND $OUT[4039] THEN
            PREVSTEP = $APP_INT[5]
            $APP_INT[5] = 185
         ENDIF
      ;ENDFOLD
      ;FOLD Schritt 188 = !E2115 & E2116 & A4039  ;%{SE}%MKUKATPVW %CVW_SPS %VST_CON %P 2:Schritt 188 = !E2115 & E2116 & A4039 , 3: ST_CON
         IF NOT $IN[2115] AND $IN[2116] AND $OUT[4039] THEN
            PREVSTEP = $APP_INT[5]
            $APP_INT[5] = 188
         ENDIF
      ;ENDFOLD
   ;ENDFOLD
   ;FOLD SCHRITT 185 --KL1 Spueleimer (an Pneum. Schwenkeinheit KL1)-- ;%{P}%MKUKATPVW,%CSTEP,%VST_NR,%P 1:SCHRITT, 2:185, 3:KL1 Spueleimer (an Pneum. Schwenkeinheit KL1)
      ;FOLD ;%{H}
         Case 185
      ;ENDFOLD
      ;FOLD -- Steuerluft EIN -- ;%{SE}%MKUKATPVW %CVW_COM %VCOMMENT %P 2:-- Steuerluft EIN --, 3: VW_COMMENT
      ;ENDFOLD
      ;FOLD A2113 = A4039 ;%{SE}%MKUKATPVW %CVW_SPS %VBOASG %P 2:A2113 = A4039, 3: BOASG
         $OUT[2113] = $OUT[4039]
      ;ENDFOLD
      ;FOLD -- RSK Fehlerausgabe Schwenkeinheit 1 Ruhest. -- ;%{SE}%MKUKATPVW %CVW_COM %VCOMMENT %P 2:-- RSK Fehlerausgabe Schwenkeinheit 1 Ruhest. --, 3: VW_COMMENT
      ;ENDFOLD
      ;FOLD F323 = !E2115 ;%{SE}%MKUKATPVW %CVW_SPS %VBOASG %P 2:F323 = !E2115, 3: BOASG
         $FLAG[323] = NOT $IN[2115]
      ;ENDFOLD
      ;FOLD -- RSK Sammelstoerung -- ;%{SE}%MKUKATPVW %CVW_COM %VCOMMENT %P 2:-- RSK Sammelstoerung --, 3: VW_COMMENT
      ;ENDFOLD
      ;FOLD F329 = F323 ;%{SE}%MKUKATPVW %CVW_SPS %VBOASG %P 2:F329 = F323, 3: BOASG
         $FLAG[329] = $FLAG[323]
      ;ENDFOLD
      ;FOLD Schritt 184 = (E26 + E27) & F323 & A4039  ;%{SE}%MKUKATPVW %CVW_SPS %VST_CON %P 2:Schritt 184 = (E26 + E27) & F323 & A4039 , 3: ST_CON
         IF ($IN[26] OR $IN[27]) AND $FLAG[323] AND $OUT[4039] THEN
            PREVSTEP = $APP_INT[5]
            $APP_INT[5] = 184
         ENDIF
      ;ENDFOLD
      ;FOLD Schritt 186 = (F523 & !F524 & E2113 + !F523 & F524 & !E2114) & A4039  ;%{SE}%MKUKATPVW %CVW_SPS %VST_CON %P 2:Schritt 186 = (F523 & !F524 & E2113 + !F523 & F524 & !E2114) & A4039 , 3: ST_CON
         IF ($FLAG[523] AND NOT $FLAG[524] AND $IN[2113] OR NOT $FLAG[523] AND $FLAG[524] AND NOT $IN[2114]) AND $OUT[4039] THEN
            PREVSTEP = $APP_INT[5]
            $APP_INT[5] = 186
         ENDIF
      ;ENDFOLD
   ;ENDFOLD
   ;FOLD SCHRITT 186 --KL1 Spueleimer (an Pneum. Schwenkeinheit KL1)-- ;%{P}%MKUKATPVW,%CSTEP,%VST_NR,%P 1:SCHRITT, 2:186, 3:KL1 Spueleimer (an Pneum. Schwenkeinheit KL1)
      ;FOLD ;%{H}
         Case 186
      ;ENDFOLD
      ;FOLD -- Steuerluft EIN -- ;%{SE}%MKUKATPVW %CVW_COM %VCOMMENT %P 2:-- Steuerluft EIN --, 3: VW_COMMENT
      ;ENDFOLD
      ;FOLD A2113 = A4039 ;%{SE}%MKUKATPVW %CVW_SPS %VBOASG %P 2:A2113 = A4039, 3: BOASG
         $OUT[2113] = $OUT[4039]
      ;ENDFOLD
      ;FOLD -- Schwenkeinheit 1 in Arbeitsstellung schwenken -- ;%{SE}%MKUKATPVW %CVW_COM %VCOMMENT %P 2:-- Schwenkeinheit 1 in Arbeitsstellung schwenken --, 3: VW_COMMENT
      ;ENDFOLD
      ;FOLD A2115 = AUS ;%{SE}%MKUKATPVW %CVW_SPS %VBOASG %P 2:A2115 = AUS, 3: BOASG
         $OUT[2115] = FALSE
      ;ENDFOLD
      ;FOLD A2116 = EIN ;%{SE}%MKUKATPVW %CVW_SPS %VBOASG %P 2:A2116 = EIN, 3: BOASG
         $OUT[2116] = TRUE
      ;ENDFOLD
      ;FOLD -- FRG Bewegung EIN -- ;%{SE}%MKUKATPVW %CVW_COM %VCOMMENT %P 2:-- FRG Bewegung EIN --, 3: VW_COMMENT
      ;ENDFOLD
      ;FOLD A2117 = AUS ;%{SE}%MKUKATPVW %CVW_SPS %VBOASG %P 2:A2117 = AUS, 3: BOASG
         $OUT[2117] = FALSE
      ;ENDFOLD
      ;FOLD A2118 = EIN ;%{SE}%MKUKATPVW %CVW_SPS %VBOASG %P 2:A2118 = EIN, 3: BOASG
         $OUT[2118] = TRUE
      ;ENDFOLD
      ;FOLD Schritt 187 = !E2115 & E2116 & A4039 + T8  ;%{SE}%MKUKATPVW %CVW_SPS %VST_CON %P 2:Schritt 187 = !E2115 & E2116 & A4039 + T8 , 3: ST_CON
         IF NOT $IN[2115] AND $IN[2116] AND $OUT[4039] OR $TIMER_FLAG[8] THEN
            PREVSTEP = $APP_INT[5]
            $APP_INT[5] = 187
         ENDIF
      ;ENDFOLD
   ;ENDFOLD
   ;FOLD SCHRITT 187 --KL1 Spueleimer (an Pneum. Schwenkeinheit KL1)-- ;%{P}%MKUKATPVW,%CSTEP,%VST_NR,%P 1:SCHRITT, 2:187, 3:KL1 Spueleimer (an Pneum. Schwenkeinheit KL1)
      ;FOLD ;%{H}
         Case 187
      ;ENDFOLD
      ;FOLD -- Steuerluft EIN -- ;%{SE}%MKUKATPVW %CVW_COM %VCOMMENT %P 2:-- Steuerluft EIN --, 3: VW_COMMENT
      ;ENDFOLD
      ;FOLD A2113 = A4039 ;%{SE}%MKUKATPVW %CVW_SPS %VBOASG %P 2:A2113 = A4039, 3: BOASG
         $OUT[2113] = $OUT[4039]
      ;ENDFOLD
      ;FOLD -- RSK Fehlerausgabe Schwenkeinheit 1 Arbeitsstellung -- ;%{SE}%MKUKATPVW %CVW_COM %VCOMMENT %P 2:-- RSK Fehlerausgabe Schwenkeinheit 1 Arbeitsstellung --, 3: VW_COMMENT
      ;ENDFOLD
      ;FOLD F324 = !E2116 & T8 + F324 ;%{SE}%MKUKATPVW %CVW_SPS %VBOASG %P 2:F324 = !E2116 & T8 + F324, 3: BOASG
         $FLAG[324] = NOT $IN[2116] AND $TIMER_FLAG[8] OR $FLAG[324]
      ;ENDFOLD
      ;FOLD -- RSK Sammelstoerung -- ;%{SE}%MKUKATPVW %CVW_COM %VCOMMENT %P 2:-- RSK Sammelstoerung --, 3: VW_COMMENT
      ;ENDFOLD
      ;FOLD F329 = F324 ;%{SE}%MKUKATPVW %CVW_SPS %VBOASG %P 2:F329 = F324, 3: BOASG
         $FLAG[329] = $FLAG[324]
      ;ENDFOLD
      ;FOLD A2116 = AUS ;%{SE}%MKUKATPVW %CVW_SPS %VBOASG %P 2:A2116 = AUS, 3: BOASG
         $OUT[2116] = FALSE
      ;ENDFOLD
      ;FOLD -- FRG Bewegung AUS -- ;%{SE}%MKUKATPVW %CVW_COM %VCOMMENT %P 2:-- FRG Bewegung AUS --, 3: VW_COMMENT
      ;ENDFOLD
      ;FOLD A2118 = AUS ;%{SE}%MKUKATPVW %CVW_SPS %VBOASG %P 2:A2118 = AUS, 3: BOASG
         $OUT[2118] = FALSE
      ;ENDFOLD
      ;FOLD Schritt 184 = F324 & (E26 + E27) & A4039  ;%{SE}%MKUKATPVW %CVW_SPS %VST_CON %P 2:Schritt 184 = F324 & (E26 + E27) & A4039 , 3: ST_CON
         IF $FLAG[324] AND ($IN[26] OR $IN[27]) AND $OUT[4039] THEN
            PREVSTEP = $APP_INT[5]
            $APP_INT[5] = 184
         ENDIF
      ;ENDFOLD
      ;FOLD Schritt 188 = !F324 & (E2118 + F837) & A4039  ;%{SE}%MKUKATPVW %CVW_SPS %VST_CON %P 2:Schritt 188 = !F324 & (E2118 + F837) & A4039 , 3: ST_CON
         IF NOT $FLAG[324] AND ($IN[2118] OR $FLAG[837]) AND $OUT[4039] THEN
            PREVSTEP = $APP_INT[5]
            $APP_INT[5] = 188
         ENDIF
      ;ENDFOLD
   ;ENDFOLD
   ;FOLD SCHRITT 188 --KL1 Spueleimer (an Pneum. Schwenkeinheit KL1)-- ;%{P}%MKUKATPVW,%CSTEP,%VST_NR,%P 1:SCHRITT, 2:188, 3:KL1 Spueleimer (an Pneum. Schwenkeinheit KL1)
      ;FOLD ;%{H}
         Case 188
      ;ENDFOLD
      ;FOLD -- Steuerluft EIN -- ;%{SE}%MKUKATPVW %CVW_COM %VCOMMENT %P 2:-- Steuerluft EIN --, 3: VW_COMMENT
      ;ENDFOLD
      ;FOLD A2113 = A4039 ;%{SE}%MKUKATPVW %CVW_SPS %VBOASG %P 2:A2113 = A4039, 3: BOASG
         $OUT[2113] = $OUT[4039]
      ;ENDFOLD
      ;FOLD -- RSK Sammelstoerung -- ;%{SE}%MKUKATPVW %CVW_COM %VCOMMENT %P 2:-- RSK Sammelstoerung --, 3: VW_COMMENT
      ;ENDFOLD
      ;FOLD F329 = T8 ;%{SE}%MKUKATPVW %CVW_SPS %VBOASG %P 2:F329 = T8, 3: BOASG
         $FLAG[329] = $TIMER_FLAG[8]
      ;ENDFOLD
      ;FOLD -- FRG in Endlage halten ein -- ;%{SE}%MKUKATPVW %CVW_COM %VCOMMENT %P 2:-- FRG in Endlage halten ein --, 3: VW_COMMENT
      ;ENDFOLD
      ;FOLD A2117 = EIN ;%{SE}%MKUKATPVW %CVW_SPS %VBOASG %P 2:A2117 = EIN, 3: BOASG
         $OUT[2117] = TRUE
      ;ENDFOLD
      ;FOLD A161 = AUS ;%{SE}%MKUKATPVW %CVW_SPS %VBOASG %P 2:A161 = AUS, 3: BOASG
         $OUT[161] = FALSE
      ;ENDFOLD
      ;FOLD t8 ( EIN ) = STOP ;%{SE}%MKUKATPVW %CVW_SPS %VTSTOP %P 2:t8 ( EIN ) = STOP, 3: TSTOP
         VW(#SET_TIME,TRUE,8,1,0)
      ;ENDFOLD
      ;FOLD F355 = !E2115 & E2116 ;%{SE}%MKUKATPVW %CVW_SPS %VBOASG %P 2:F355 = !E2115 & E2116, 3: BOASG
         $FLAG[355] = NOT $IN[2115] AND $IN[2116]
      ;ENDFOLD
      ;FOLD Schritt 1 = !E2117 & (E2118 + F837) & F355 & A4039  ;%{SE}%MKUKATPVW %CVW_SPS %VST_CON %P 2:Schritt 1 = !E2117 & (E2118 + F837) & F355 & A4039 , 3: ST_CON
         IF NOT $IN[2117] AND ($IN[2118] OR $FLAG[837]) AND $FLAG[355] AND $OUT[4039] THEN
            PREVSTEP = $APP_INT[5]
            $APP_INT[5] = 1
         ENDIF
      ;ENDFOLD
   ;ENDFOLD
   ;FOLD SCHRITT 189 --KL1 Spueleimer (an Pneum. Schwenkeinheit KL1)-- ;%{P}%MKUKATPVW,%CSTEP,%VST_NR,%P 1:SCHRITT, 2:189, 3:KL1 Spueleimer (an Pneum. Schwenkeinheit KL1)
      ;FOLD ;%{H}
         Case 189
      ;ENDFOLD
      ;FOLD -- Steuerluft EIN -- ;%{SE}%MKUKATPVW %CVW_COM %VCOMMENT %P 2:-- Steuerluft EIN --, 3: VW_COMMENT
      ;ENDFOLD
      ;FOLD A2113 = A4039 ;%{SE}%MKUKATPVW %CVW_SPS %VBOASG %P 2:A2113 = A4039, 3: BOASG
         $OUT[2113] = $OUT[4039]
      ;ENDFOLD
      ;FOLD -- RSK gestartet -- ;%{SE}%MKUKATPVW %CVW_COM %VCOMMENT %P 2:-- RSK gestartet --, 3: VW_COMMENT
      ;ENDFOLD
      ;FOLD F321 = AUS ;%{SE}%MKUKATPVW %CVW_SPS %VBOASG %P 2:F321 = AUS, 3: BOASG
         $FLAG[321] = FALSE
      ;ENDFOLD
      ;FOLD F323 = AUS ;%{SE}%MKUKATPVW %CVW_SPS %VBOASG %P 2:F323 = AUS, 3: BOASG
         $FLAG[323] = FALSE
      ;ENDFOLD
      ;FOLD F324 = AUS ;%{SE}%MKUKATPVW %CVW_SPS %VBOASG %P 2:F324 = AUS, 3: BOASG
         $FLAG[324] = FALSE
      ;ENDFOLD
      ;FOLD F329 = AUS ;%{SE}%MKUKATPVW %CVW_SPS %VBOASG %P 2:F329 = AUS, 3: BOASG
         $FLAG[329] = FALSE
      ;ENDFOLD
      ;FOLD A161 = EIN ;%{SE}%MKUKATPVW %CVW_SPS %VBOASG %P 2:A161 = EIN, 3: BOASG
         $OUT[161] = TRUE
      ;ENDFOLD
      ;FOLD A2115 = AUS ;%{SE}%MKUKATPVW %CVW_SPS %VBOASG %P 2:A2115 = AUS, 3: BOASG
         $OUT[2115] = FALSE
      ;ENDFOLD
      ;FOLD A2116 = AUS ;%{SE}%MKUKATPVW %CVW_SPS %VBOASG %P 2:A2116 = AUS, 3: BOASG
         $OUT[2116] = FALSE
      ;ENDFOLD
      ;FOLD A2117 = AUS ;%{SE}%MKUKATPVW %CVW_SPS %VBOASG %P 2:A2117 = AUS, 3: BOASG
         $OUT[2117] = FALSE
      ;ENDFOLD
      ;FOLD A2118 = AUS ;%{SE}%MKUKATPVW %CVW_SPS %VBOASG %P 2:A2118 = AUS, 3: BOASG
         $OUT[2118] = FALSE
      ;ENDFOLD
      ;FOLD -- Ueberwachungszeit Schwenkeinheit 1 schwenken -- ;%{SE}%MKUKATPVW %CVW_COM %VCOMMENT %P 2:-- Ueberwachungszeit Schwenkeinheit 1 schwenken --, 3: VW_COMMENT
      ;ENDFOLD
      ;FOLD t8 ( EIN ) = -100[1/10Sek] ;%{SE}%MKUKATPVW %CVW_SPS %VTASG %P 2:t8 ( EIN ) = -100[1/10Sek], 3: TASG
         VW(#SET_TIME,TRUE,8,0,-100)
      ;ENDFOLD
      ;FOLD Schritt 190 = !E2115 & A4039  ;%{SE}%MKUKATPVW %CVW_SPS %VST_CON %P 2:Schritt 190 = !E2115 & A4039 , 3: ST_CON
         IF NOT $IN[2115] AND $OUT[4039] THEN
            PREVSTEP = $APP_INT[5]
            $APP_INT[5] = 190
         ENDIF
      ;ENDFOLD
      ;FOLD Schritt 193 = E2115 & !E2116 & A4039  ;%{SE}%MKUKATPVW %CVW_SPS %VST_CON %P 2:Schritt 193 = E2115 & !E2116 & A4039 , 3: ST_CON
         IF $IN[2115] AND NOT $IN[2116] AND $OUT[4039] THEN
            PREVSTEP = $APP_INT[5]
            $APP_INT[5] = 193
         ENDIF
      ;ENDFOLD
   ;ENDFOLD
   ;FOLD SCHRITT 190 --KL1 Spueleimer (an Pneum. Schwenkeinheit KL1)-- ;%{P}%MKUKATPVW,%CSTEP,%VST_NR,%P 1:SCHRITT, 2:190, 3:KL1 Spueleimer (an Pneum. Schwenkeinheit KL1)
      ;FOLD ;%{H}
         Case 190
      ;ENDFOLD
      ;FOLD -- Steuerluft EIN -- ;%{SE}%MKUKATPVW %CVW_COM %VCOMMENT %P 2:-- Steuerluft EIN --, 3: VW_COMMENT
      ;ENDFOLD
      ;FOLD A2113 = A4039 ;%{SE}%MKUKATPVW %CVW_SPS %VBOASG %P 2:A2113 = A4039, 3: BOASG
         $OUT[2113] = $OUT[4039]
      ;ENDFOLD
      ;FOLD -- RSK Fehlerausgabe Schwenkeinheit 1 Arbeit. -- ;%{SE}%MKUKATPVW %CVW_COM %VCOMMENT %P 2:-- RSK Fehlerausgabe Schwenkeinheit 1 Arbeit. --, 3: VW_COMMENT
      ;ENDFOLD
      ;FOLD F324 = !E2116 ;%{SE}%MKUKATPVW %CVW_SPS %VBOASG %P 2:F324 = !E2116, 3: BOASG
         $FLAG[324] = NOT $IN[2116]
      ;ENDFOLD
      ;FOLD -- RSK Sammelstoerung -- ;%{SE}%MKUKATPVW %CVW_COM %VCOMMENT %P 2:-- RSK Sammelstoerung --, 3: VW_COMMENT
      ;ENDFOLD
      ;FOLD F329 = F324 ;%{SE}%MKUKATPVW %CVW_SPS %VBOASG %P 2:F329 = F324, 3: BOASG
         $FLAG[329] = $FLAG[324]
      ;ENDFOLD
      ;FOLD Schritt 189 = (E26 + E27) & F324 & A4039  ;%{SE}%MKUKATPVW %CVW_SPS %VST_CON %P 2:Schritt 189 = (E26 + E27) & F324 & A4039 , 3: ST_CON
         IF ($IN[26] OR $IN[27]) AND $FLAG[324] AND $OUT[4039] THEN
            PREVSTEP = $APP_INT[5]
            $APP_INT[5] = 189
         ENDIF
      ;ENDFOLD
      ;FOLD Schritt 191 = (F523 & !F524 & E2113 + !F523 & F524 & !E2114) & A4039  ;%{SE}%MKUKATPVW %CVW_SPS %VST_CON %P 2:Schritt 191 = (F523 & !F524 & E2113 + !F523 & F524 & !E2114) & A4039 , 3: ST_CON
         IF ($FLAG[523] AND NOT $FLAG[524] AND $IN[2113] OR NOT $FLAG[523] AND $FLAG[524] AND NOT $IN[2114]) AND $OUT[4039] THEN
            PREVSTEP = $APP_INT[5]
            $APP_INT[5] = 191
         ENDIF
      ;ENDFOLD
   ;ENDFOLD
   ;FOLD SCHRITT 191 --KL1 Spueleimer (an Pneum. Schwenkeinheit KL1)-- ;%{P}%MKUKATPVW,%CSTEP,%VST_NR,%P 1:SCHRITT, 2:191, 3:KL1 Spueleimer (an Pneum. Schwenkeinheit KL1)
      ;FOLD ;%{H}
         Case 191
      ;ENDFOLD
      ;FOLD -- Steuerluft EIN -- ;%{SE}%MKUKATPVW %CVW_COM %VCOMMENT %P 2:-- Steuerluft EIN --, 3: VW_COMMENT
      ;ENDFOLD
      ;FOLD A2113 = A4039 ;%{SE}%MKUKATPVW %CVW_SPS %VBOASG %P 2:A2113 = A4039, 3: BOASG
         $OUT[2113] = $OUT[4039]
      ;ENDFOLD
      ;FOLD -- Schwenkeinheit 1 in Ruhestellung schwenken -- ;%{SE}%MKUKATPVW %CVW_COM %VCOMMENT %P 2:-- Schwenkeinheit 1 in Ruhestellung schwenken --, 3: VW_COMMENT
      ;ENDFOLD
      ;FOLD A2115 = EIN ;%{SE}%MKUKATPVW %CVW_SPS %VBOASG %P 2:A2115 = EIN, 3: BOASG
         $OUT[2115] = TRUE
      ;ENDFOLD
      ;FOLD A2116 = AUS ;%{SE}%MKUKATPVW %CVW_SPS %VBOASG %P 2:A2116 = AUS, 3: BOASG
         $OUT[2116] = FALSE
      ;ENDFOLD
      ;FOLD -- FRG Bewegung EIN -- ;%{SE}%MKUKATPVW %CVW_COM %VCOMMENT %P 2:-- FRG Bewegung EIN --, 3: VW_COMMENT
      ;ENDFOLD
      ;FOLD A2117 = AUS ;%{SE}%MKUKATPVW %CVW_SPS %VBOASG %P 2:A2117 = AUS, 3: BOASG
         $OUT[2117] = FALSE
      ;ENDFOLD
      ;FOLD A2118 = EIN ;%{SE}%MKUKATPVW %CVW_SPS %VBOASG %P 2:A2118 = EIN, 3: BOASG
         $OUT[2118] = TRUE
      ;ENDFOLD
      ;FOLD Schritt 192 = E2115 & !E2116 & A4039 + T8  ;%{SE}%MKUKATPVW %CVW_SPS %VST_CON %P 2:Schritt 192 = E2115 & !E2116 & A4039 + T8 , 3: ST_CON
         IF $IN[2115] AND NOT $IN[2116] AND $OUT[4039] OR $TIMER_FLAG[8] THEN
            PREVSTEP = $APP_INT[5]
            $APP_INT[5] = 192
         ENDIF
      ;ENDFOLD
   ;ENDFOLD
   ;FOLD SCHRITT 192 --KL1 Spueleimer (an Pneum. Schwenkeinheit KL1)-- ;%{P}%MKUKATPVW,%CSTEP,%VST_NR,%P 1:SCHRITT, 2:192, 3:KL1 Spueleimer (an Pneum. Schwenkeinheit KL1)
      ;FOLD ;%{H}
         Case 192
      ;ENDFOLD
      ;FOLD -- Steuerluft EIN -- ;%{SE}%MKUKATPVW %CVW_COM %VCOMMENT %P 2:-- Steuerluft EIN --, 3: VW_COMMENT
      ;ENDFOLD
      ;FOLD A2113 = A4039 ;%{SE}%MKUKATPVW %CVW_SPS %VBOASG %P 2:A2113 = A4039, 3: BOASG
         $OUT[2113] = $OUT[4039]
      ;ENDFOLD
      ;FOLD -- RSK Fehlerausgabe Schwenkeinheit 1 Ruhestellung -- ;%{SE}%MKUKATPVW %CVW_COM %VCOMMENT %P 2:-- RSK Fehlerausgabe Schwenkeinheit 1 Ruhestellung --, 3: VW_COMMENT
      ;ENDFOLD
      ;FOLD F323 = !E2115 & T8 + F323 ;%{SE}%MKUKATPVW %CVW_SPS %VBOASG %P 2:F323 = !E2115 & T8 + F323, 3: BOASG
         $FLAG[323] = NOT $IN[2115] AND $TIMER_FLAG[8] OR $FLAG[323]
      ;ENDFOLD
      ;FOLD -- RSK Sammelstoerung -- ;%{SE}%MKUKATPVW %CVW_COM %VCOMMENT %P 2:-- RSK Sammelstoerung --, 3: VW_COMMENT
      ;ENDFOLD
      ;FOLD F329 = F323 ;%{SE}%MKUKATPVW %CVW_SPS %VBOASG %P 2:F329 = F323, 3: BOASG
         $FLAG[329] = $FLAG[323]
      ;ENDFOLD
      ;FOLD A2115 = AUS ;%{SE}%MKUKATPVW %CVW_SPS %VBOASG %P 2:A2115 = AUS, 3: BOASG
         $OUT[2115] = FALSE
      ;ENDFOLD
      ;FOLD -- FRG Bewegung AUS -- ;%{SE}%MKUKATPVW %CVW_COM %VCOMMENT %P 2:-- FRG Bewegung AUS --, 3: VW_COMMENT
      ;ENDFOLD
      ;FOLD A2118 = AUS ;%{SE}%MKUKATPVW %CVW_SPS %VBOASG %P 2:A2118 = AUS, 3: BOASG
         $OUT[2118] = FALSE
      ;ENDFOLD
      ;FOLD Schritt 189 = F323 & (E26 + E27) & A4039  ;%{SE}%MKUKATPVW %CVW_SPS %VST_CON %P 2:Schritt 189 = F323 & (E26 + E27) & A4039 , 3: ST_CON
         IF $FLAG[323] AND ($IN[26] OR $IN[27]) AND $OUT[4039] THEN
            PREVSTEP = $APP_INT[5]
            $APP_INT[5] = 189
         ENDIF
      ;ENDFOLD
      ;FOLD Schritt 193 = !F323 & (E2118 + F837) & A4039  ;%{SE}%MKUKATPVW %CVW_SPS %VST_CON %P 2:Schritt 193 = !F323 & (E2118 + F837) & A4039 , 3: ST_CON
         IF NOT $FLAG[323] AND ($IN[2118] OR $FLAG[837]) AND $OUT[4039] THEN
            PREVSTEP = $APP_INT[5]
            $APP_INT[5] = 193
         ENDIF
      ;ENDFOLD
   ;ENDFOLD
   ;FOLD SCHRITT 193 --KL1 Spueleimer (an Pneum. Schwenkeinheit KL1)-- ;%{P}%MKUKATPVW,%CSTEP,%VST_NR,%P 1:SCHRITT, 2:193, 3:KL1 Spueleimer (an Pneum. Schwenkeinheit KL1)
      ;FOLD ;%{H}
         Case 193
      ;ENDFOLD
      ;FOLD -- Steuerluft EIN -- ;%{SE}%MKUKATPVW %CVW_COM %VCOMMENT %P 2:-- Steuerluft EIN --, 3: VW_COMMENT
      ;ENDFOLD
      ;FOLD A2113 = A4039 ;%{SE}%MKUKATPVW %CVW_SPS %VBOASG %P 2:A2113 = A4039, 3: BOASG
         $OUT[2113] = $OUT[4039]
      ;ENDFOLD
      ;FOLD F323 = AUS ;%{SE}%MKUKATPVW %CVW_SPS %VBOASG %P 2:F323 = AUS, 3: BOASG
         $FLAG[323] = FALSE
      ;ENDFOLD
      ;FOLD F329 = T8 ;%{SE}%MKUKATPVW %CVW_SPS %VBOASG %P 2:F329 = T8, 3: BOASG
         $FLAG[329] = $TIMER_FLAG[8]
      ;ENDFOLD
      ;FOLD -- FRG in Endlage halten ein -- ;%{SE}%MKUKATPVW %CVW_COM %VCOMMENT %P 2:-- FRG in Endlage halten ein --, 3: VW_COMMENT
      ;ENDFOLD
      ;FOLD A2117 = EIN ;%{SE}%MKUKATPVW %CVW_SPS %VBOASG %P 2:A2117 = EIN, 3: BOASG
         $OUT[2117] = TRUE
      ;ENDFOLD
      ;FOLD Schritt 194 = !E2117 & (E2118 + F837) & A4039  ;%{SE}%MKUKATPVW %CVW_SPS %VST_CON %P 2:Schritt 194 = !E2117 & (E2118 + F837) & A4039 , 3: ST_CON
         IF NOT $IN[2117] AND ($IN[2118] OR $FLAG[837]) AND $OUT[4039] THEN
            PREVSTEP = $APP_INT[5]
            $APP_INT[5] = 194
         ENDIF
      ;ENDFOLD
   ;ENDFOLD
   ;FOLD SCHRITT 194 --KL1 Spueleimer (an Pneum. Schwenkeinheit KL1)-- ;%{P}%MKUKATPVW,%CSTEP,%VST_NR,%P 1:SCHRITT, 2:194, 3:KL1 Spueleimer (an Pneum. Schwenkeinheit KL1)
      ;FOLD ;%{H}
         Case 194
      ;ENDFOLD
      ;FOLD -- Steuerluft EIN -- ;%{SE}%MKUKATPVW %CVW_COM %VCOMMENT %P 2:-- Steuerluft EIN --, 3: VW_COMMENT
      ;ENDFOLD
      ;FOLD A2113 = A4039 ;%{SE}%MKUKATPVW %CVW_SPS %VBOASG %P 2:A2113 = A4039, 3: BOASG
         $OUT[2113] = $OUT[4039]
      ;ENDFOLD
      ;FOLD -- RSK Sammelstoerung -- ;%{SE}%MKUKATPVW %CVW_COM %VCOMMENT %P 2:-- RSK Sammelstoerung --, 3: VW_COMMENT
      ;ENDFOLD
      ;FOLD F329 = T8 ;%{SE}%MKUKATPVW %CVW_SPS %VBOASG %P 2:F329 = T8, 3: BOASG
         $FLAG[329] = $TIMER_FLAG[8]
      ;ENDFOLD
      ;FOLD -- FRG in Endlage halten AUS -- ;%{SE}%MKUKATPVW %CVW_COM %VCOMMENT %P 2:-- FRG in Endlage halten AUS --, 3: VW_COMMENT
      ;ENDFOLD
      ;FOLD A2117 = AUS ;%{SE}%MKUKATPVW %CVW_SPS %VBOASG %P 2:A2117 = AUS, 3: BOASG
         $OUT[2117] = FALSE
      ;ENDFOLD
      ;FOLD A161 = AUS ;%{SE}%MKUKATPVW %CVW_SPS %VBOASG %P 2:A161 = AUS, 3: BOASG
         $OUT[161] = FALSE
      ;ENDFOLD
      ;FOLD t8 ( EIN ) = STOP ;%{SE}%MKUKATPVW %CVW_SPS %VTSTOP %P 2:t8 ( EIN ) = STOP, 3: TSTOP
         VW(#SET_TIME,TRUE,8,1,0)
      ;ENDFOLD
      ;FOLD F355 = E2115 & !E2116 ;%{SE}%MKUKATPVW %CVW_SPS %VBOASG %P 2:F355 = E2115 & !E2116, 3: BOASG
         $FLAG[355] = $IN[2115] AND NOT $IN[2116]
      ;ENDFOLD
      ;FOLD Schritt 1 = F355 & A4039  ;%{SE}%MKUKATPVW %CVW_SPS %VST_CON %P 2:Schritt 1 = F355 & A4039 , 3: ST_CON
         IF $FLAG[355] AND $OUT[4039] THEN
            PREVSTEP = $APP_INT[5]
            $APP_INT[5] = 1
         ENDIF
      ;ENDFOLD
   ;ENDFOLD
   ;FOLD SCHRITT 195 --KL2 Spueleimer (an Pneum. Schwenkeinheit KL2)-- ;%{P}%MKUKATPVW,%CSTEP,%VST_NR,%P 1:SCHRITT, 2:195, 3:KL2 Spueleimer (an Pneum. Schwenkeinheit KL2)
      ;FOLD ;%{H}
         Case 195
      ;ENDFOLD
      ;FOLD -- RSK gestartet -- ;%{SE}%MKUKATPVW %CVW_COM %VCOMMENT %P 2:-- RSK gestartet --, 3: VW_COMMENT
      ;ENDFOLD
      ;FOLD F321 = AUS ;%{SE}%MKUKATPVW %CVW_SPS %VBOASG %P 2:F321 = AUS, 3: BOASG
         $FLAG[321] = FALSE
      ;ENDFOLD
      ;FOLD F323 = AUS ;%{SE}%MKUKATPVW %CVW_SPS %VBOASG %P 2:F323 = AUS, 3: BOASG
         $FLAG[323] = FALSE
      ;ENDFOLD
      ;FOLD F324 = AUS ;%{SE}%MKUKATPVW %CVW_SPS %VBOASG %P 2:F324 = AUS, 3: BOASG
         $FLAG[324] = FALSE
      ;ENDFOLD
      ;FOLD F329 = AUS ;%{SE}%MKUKATPVW %CVW_SPS %VBOASG %P 2:F329 = AUS, 3: BOASG
         $FLAG[329] = FALSE
      ;ENDFOLD
      ;FOLD A177 = EIN ;%{SE}%MKUKATPVW %CVW_SPS %VBOASG %P 2:A177 = EIN, 3: BOASG
         $OUT[177] = TRUE
      ;ENDFOLD
      ;FOLD -- Steuerluft EIN -- ;%{SE}%MKUKATPVW %CVW_COM %VCOMMENT %P 2:-- Steuerluft EIN --, 3: VW_COMMENT
      ;ENDFOLD
      ;FOLD A2121 = A4039 ;%{SE}%MKUKATPVW %CVW_SPS %VBOASG %P 2:A2121 = A4039, 3: BOASG
         $OUT[2121] = $OUT[4039]
      ;ENDFOLD
      ;FOLD A2123 = AUS ;%{SE}%MKUKATPVW %CVW_SPS %VBOASG %P 2:A2123 = AUS, 3: BOASG
         $OUT[2123] = FALSE
      ;ENDFOLD
      ;FOLD A2124 = AUS ;%{SE}%MKUKATPVW %CVW_SPS %VBOASG %P 2:A2124 = AUS, 3: BOASG
         $OUT[2124] = FALSE
      ;ENDFOLD
      ;FOLD A2125 = AUS ;%{SE}%MKUKATPVW %CVW_SPS %VBOASG %P 2:A2125 = AUS, 3: BOASG
         $OUT[2125] = FALSE
      ;ENDFOLD
      ;FOLD A2126 = AUS ;%{SE}%MKUKATPVW %CVW_SPS %VBOASG %P 2:A2126 = AUS, 3: BOASG
         $OUT[2126] = FALSE
      ;ENDFOLD
      ;FOLD -- Ueberwachungszeit Schwenkeinheit 2 -- ;%{SE}%MKUKATPVW %CVW_COM %VCOMMENT %P 2:-- Ueberwachungszeit Schwenkeinheit 2 --, 3: VW_COMMENT
      ;ENDFOLD
      ;FOLD t8 ( EIN ) = -100[1/10Sek] ;%{SE}%MKUKATPVW %CVW_SPS %VTASG %P 2:t8 ( EIN ) = -100[1/10Sek], 3: TASG
         VW(#SET_TIME,TRUE,8,0,-100)
      ;ENDFOLD
      ;FOLD Schritt 196 = !E2124 & A4039  ;%{SE}%MKUKATPVW %CVW_SPS %VST_CON %P 2:Schritt 196 = !E2124 & A4039 , 3: ST_CON
         IF NOT $IN[2124] AND $OUT[4039] THEN
            PREVSTEP = $APP_INT[5]
            $APP_INT[5] = 196
         ENDIF
      ;ENDFOLD
      ;FOLD Schritt 199 = !E2123 & E2124 & A4039  ;%{SE}%MKUKATPVW %CVW_SPS %VST_CON %P 2:Schritt 199 = !E2123 & E2124 & A4039 , 3: ST_CON
         IF NOT $IN[2123] AND $IN[2124] AND $OUT[4039] THEN
            PREVSTEP = $APP_INT[5]
            $APP_INT[5] = 199
         ENDIF
      ;ENDFOLD
   ;ENDFOLD
   ;FOLD SCHRITT 196 --KL2 Spueleimer (an Pneum. Schwenkeinheit KL2)-- ;%{P}%MKUKATPVW,%CSTEP,%VST_NR,%P 1:SCHRITT, 2:196, 3:KL2 Spueleimer (an Pneum. Schwenkeinheit KL2)
      ;FOLD ;%{H}
         Case 196
      ;ENDFOLD
      ;FOLD -- Steuerluft EIN -- ;%{SE}%MKUKATPVW %CVW_COM %VCOMMENT %P 2:-- Steuerluft EIN --, 3: VW_COMMENT
      ;ENDFOLD
      ;FOLD A2121 = A4039 ;%{SE}%MKUKATPVW %CVW_SPS %VBOASG %P 2:A2121 = A4039, 3: BOASG
         $OUT[2121] = $OUT[4039]
      ;ENDFOLD
      ;FOLD -- RSK Fehlerausgabe Schwenkeinheit 2 Ruhest. -- ;%{SE}%MKUKATPVW %CVW_COM %VCOMMENT %P 2:-- RSK Fehlerausgabe Schwenkeinheit 2 Ruhest. --, 3: VW_COMMENT
      ;ENDFOLD
      ;FOLD F323 = !E2123 ;%{SE}%MKUKATPVW %CVW_SPS %VBOASG %P 2:F323 = !E2123, 3: BOASG
         $FLAG[323] = NOT $IN[2123]
      ;ENDFOLD
      ;FOLD -- RSK Sammelstoerung -- ;%{SE}%MKUKATPVW %CVW_COM %VCOMMENT %P 2:-- RSK Sammelstoerung --, 3: VW_COMMENT
      ;ENDFOLD
      ;FOLD F329 = F323 ;%{SE}%MKUKATPVW %CVW_SPS %VBOASG %P 2:F329 = F323, 3: BOASG
         $FLAG[329] = $FLAG[323]
      ;ENDFOLD
      ;FOLD Schritt 195 = (E26 + E27) & F323 & A4039  ;%{SE}%MKUKATPVW %CVW_SPS %VST_CON %P 2:Schritt 195 = (E26 + E27) & F323 & A4039 , 3: ST_CON
         IF ($IN[26] OR $IN[27]) AND $FLAG[323] AND $OUT[4039] THEN
            PREVSTEP = $APP_INT[5]
            $APP_INT[5] = 195
         ENDIF
      ;ENDFOLD
      ;FOLD Schritt 197 = (F523 & !F524 & E2121 + !F523 & F524 & !E2122) & A4039  ;%{SE}%MKUKATPVW %CVW_SPS %VST_CON %P 2:Schritt 197 = (F523 & !F524 & E2121 + !F523 & F524 & !E2122) & A4039 , 3: ST_CON
         IF ($FLAG[523] AND NOT $FLAG[524] AND $IN[2121] OR NOT $FLAG[523] AND $FLAG[524] AND NOT $IN[2122]) AND $OUT[4039] THEN
            PREVSTEP = $APP_INT[5]
            $APP_INT[5] = 197
         ENDIF
      ;ENDFOLD
   ;ENDFOLD
   ;FOLD SCHRITT 197 -- KL2 Spueleimer (an Pneum. Schwenkeinheit KL2)-- ;%{P}%MKUKATPVW,%CSTEP,%VST_NR,%P 1:SCHRITT, 2:197, 3: KL2 Spueleimer (an Pneum. Schwenkeinheit KL2)
      ;FOLD ;%{H}
         Case 197
      ;ENDFOLD
      ;FOLD -- Steuerluft EIN -- ;%{SE}%MKUKATPVW %CVW_COM %VCOMMENT %P 2:-- Steuerluft EIN --, 3: VW_COMMENT
      ;ENDFOLD
      ;FOLD A2121 = A4039 ;%{SE}%MKUKATPVW %CVW_SPS %VBOASG %P 2:A2121 = A4039, 3: BOASG
         $OUT[2121] = $OUT[4039]
      ;ENDFOLD
      ;FOLD -- Schwenkeinheit 2 in Arbeitsstellung schwenken -- ;%{SE}%MKUKATPVW %CVW_COM %VCOMMENT %P 2:-- Schwenkeinheit 2 in Arbeitsstellung schwenken --, 3: VW_COMMENT
      ;ENDFOLD
      ;FOLD A2123 = AUS ;%{SE}%MKUKATPVW %CVW_SPS %VBOASG %P 2:A2123 = AUS, 3: BOASG
         $OUT[2123] = FALSE
      ;ENDFOLD
      ;FOLD A2124 = EIN ;%{SE}%MKUKATPVW %CVW_SPS %VBOASG %P 2:A2124 = EIN, 3: BOASG
         $OUT[2124] = TRUE
      ;ENDFOLD
      ;FOLD -- FRG Bewegung EIN -- ;%{SE}%MKUKATPVW %CVW_COM %VCOMMENT %P 2:-- FRG Bewegung EIN --, 3: VW_COMMENT
      ;ENDFOLD
      ;FOLD A2125 = AUS ;%{SE}%MKUKATPVW %CVW_SPS %VBOASG %P 2:A2125 = AUS, 3: BOASG
         $OUT[2125] = FALSE
      ;ENDFOLD
      ;FOLD A2126 = EIN ;%{SE}%MKUKATPVW %CVW_SPS %VBOASG %P 2:A2126 = EIN, 3: BOASG
         $OUT[2126] = TRUE
      ;ENDFOLD
      ;FOLD Schritt 198 = E2124 & !E2123 & A4039 + T8  ;%{SE}%MKUKATPVW %CVW_SPS %VST_CON %P 2:Schritt 198 = E2124 & !E2123 & A4039 + T8 , 3: ST_CON
         IF $IN[2124] AND NOT $IN[2123] AND $OUT[4039] OR $TIMER_FLAG[8] THEN
            PREVSTEP = $APP_INT[5]
            $APP_INT[5] = 198
         ENDIF
      ;ENDFOLD
   ;ENDFOLD
   ;FOLD SCHRITT 198 -- KL2 Spueleimer (an Pneum. Schwenkeinheit KL2)-- ;%{P}%MKUKATPVW,%CSTEP,%VST_NR,%P 1:SCHRITT, 2:198, 3: KL2 Spueleimer (an Pneum. Schwenkeinheit KL2)
      ;FOLD ;%{H}
         Case 198
      ;ENDFOLD
      ;FOLD -- Steuerluft EIN -- ;%{SE}%MKUKATPVW %CVW_COM %VCOMMENT %P 2:-- Steuerluft EIN --, 3: VW_COMMENT
      ;ENDFOLD
      ;FOLD A2121 = A4039 ;%{SE}%MKUKATPVW %CVW_SPS %VBOASG %P 2:A2121 = A4039, 3: BOASG
         $OUT[2121] = $OUT[4039]
      ;ENDFOLD
      ;FOLD -- RSK Fehlerausgabe Schwenkeinheit 2 Arbeitsstellung -- ;%{SE}%MKUKATPVW %CVW_COM %VCOMMENT %P 2:-- RSK Fehlerausgabe Schwenkeinheit 2 Arbeitsstellung --, 3: VW_COMMENT
      ;ENDFOLD
      ;FOLD F324 = !E2124 & T8 + F324 ;%{SE}%MKUKATPVW %CVW_SPS %VBOASG %P 2:F324 = !E2124 & T8 + F324, 3: BOASG
         $FLAG[324] = NOT $IN[2124] AND $TIMER_FLAG[8] OR $FLAG[324]
      ;ENDFOLD
      ;FOLD -- RSK Sammelstoerung -- ;%{SE}%MKUKATPVW %CVW_COM %VCOMMENT %P 2:-- RSK Sammelstoerung --, 3: VW_COMMENT
      ;ENDFOLD
      ;FOLD F329 = F324 ;%{SE}%MKUKATPVW %CVW_SPS %VBOASG %P 2:F329 = F324, 3: BOASG
         $FLAG[329] = $FLAG[324]
      ;ENDFOLD
      ;FOLD A2124 = AUS ;%{SE}%MKUKATPVW %CVW_SPS %VBOASG %P 2:A2124 = AUS, 3: BOASG
         $OUT[2124] = FALSE
      ;ENDFOLD
      ;FOLD -- FRG Bewegung AUS -- ;%{SE}%MKUKATPVW %CVW_COM %VCOMMENT %P 2:-- FRG Bewegung AUS --, 3: VW_COMMENT
      ;ENDFOLD
      ;FOLD A2126 = AUS ;%{SE}%MKUKATPVW %CVW_SPS %VBOASG %P 2:A2126 = AUS, 3: BOASG
         $OUT[2126] = FALSE
      ;ENDFOLD
      ;FOLD Schritt 195 = F324 & (E26 + E27) & A4039  ;%{SE}%MKUKATPVW %CVW_SPS %VST_CON %P 2:Schritt 195 = F324 & (E26 + E27) & A4039 , 3: ST_CON
         IF $FLAG[324] AND ($IN[26] OR $IN[27]) AND $OUT[4039] THEN
            PREVSTEP = $APP_INT[5]
            $APP_INT[5] = 195
         ENDIF
      ;ENDFOLD
      ;FOLD Schritt 199 = !F324 & (E2126 + F837) & A4039  ;%{SE}%MKUKATPVW %CVW_SPS %VST_CON %P 2:Schritt 199 = !F324 & (E2126 + F837) & A4039 , 3: ST_CON
         IF NOT $FLAG[324] AND ($IN[2126] OR $FLAG[837]) AND $OUT[4039] THEN
            PREVSTEP = $APP_INT[5]
            $APP_INT[5] = 199
         ENDIF
      ;ENDFOLD
   ;ENDFOLD
   ;FOLD SCHRITT 199 -- KL2 Spueleimer (an Pneum. Schwenkeinheit KL2)-- ;%{P}%MKUKATPVW,%CSTEP,%VST_NR,%P 1:SCHRITT, 2:199, 3: KL2 Spueleimer (an Pneum. Schwenkeinheit KL2)
      ;FOLD ;%{H}
         Case 199
      ;ENDFOLD
      ;FOLD -- Steuerluft EIN -- ;%{SE}%MKUKATPVW %CVW_COM %VCOMMENT %P 2:-- Steuerluft EIN --, 3: VW_COMMENT
      ;ENDFOLD
      ;FOLD A2121 = A4039 ;%{SE}%MKUKATPVW %CVW_SPS %VBOASG %P 2:A2121 = A4039, 3: BOASG
         $OUT[2121] = $OUT[4039]
      ;ENDFOLD
      ;FOLD -- RSK Sammelstoerung -- ;%{SE}%MKUKATPVW %CVW_COM %VCOMMENT %P 2:-- RSK Sammelstoerung --, 3: VW_COMMENT
      ;ENDFOLD
      ;FOLD F329 = T8 ;%{SE}%MKUKATPVW %CVW_SPS %VBOASG %P 2:F329 = T8, 3: BOASG
         $FLAG[329] = $TIMER_FLAG[8]
      ;ENDFOLD
      ;FOLD -- FRG in Endlage halten ein -- ;%{SE}%MKUKATPVW %CVW_COM %VCOMMENT %P 2:-- FRG in Endlage halten ein --, 3: VW_COMMENT
      ;ENDFOLD
      ;FOLD A2125 = EIN ;%{SE}%MKUKATPVW %CVW_SPS %VBOASG %P 2:A2125 = EIN, 3: BOASG
         $OUT[2125] = TRUE
      ;ENDFOLD
      ;FOLD A177 = AUS ;%{SE}%MKUKATPVW %CVW_SPS %VBOASG %P 2:A177 = AUS, 3: BOASG
         $OUT[177] = FALSE
      ;ENDFOLD
      ;FOLD t8 ( EIN ) = STOP ;%{SE}%MKUKATPVW %CVW_SPS %VTSTOP %P 2:t8 ( EIN ) = STOP, 3: TSTOP
         VW(#SET_TIME,TRUE,8,1,0)
      ;ENDFOLD
      ;FOLD F376 =  !E2123 & E2124 ;%{SE}%MKUKATPVW %CVW_SPS %VBOASG %P 2:F376 =  !E2123 & E2124, 3: BOASG
         $FLAG[376] = NOT $IN[2123] AND $IN[2124]
      ;ENDFOLD
      ;FOLD Schritt 1 = !E2125 & (E2126 + F837) & F376 & A4039  ;%{SE}%MKUKATPVW %CVW_SPS %VST_CON %P 2:Schritt 1 = !E2125 & (E2126 + F837) & F376 & A4039 , 3: ST_CON
         IF NOT $IN[2125] AND ($IN[2126] OR $FLAG[837]) AND $FLAG[376] AND $OUT[4039] THEN
            PREVSTEP = $APP_INT[5]
            $APP_INT[5] = 1
         ENDIF
      ;ENDFOLD
   ;ENDFOLD
   ;FOLD SCHRITT 200 --KL2 Spueleimer (an Pneum. Schwenkeinheit KL2)-- ;%{P}%MKUKATPVW,%CSTEP,%VST_NR,%P 1:SCHRITT, 2:200, 3:KL2 Spueleimer (an Pneum. Schwenkeinheit KL2)
      ;FOLD ;%{H}
         Case 200
      ;ENDFOLD
      ;FOLD -- Steuerluft EIN -- ;%{SE}%MKUKATPVW %CVW_COM %VCOMMENT %P 2:-- Steuerluft EIN --, 3: VW_COMMENT
      ;ENDFOLD
      ;FOLD A2121 = A4039 ;%{SE}%MKUKATPVW %CVW_SPS %VBOASG %P 2:A2121 = A4039, 3: BOASG
         $OUT[2121] = $OUT[4039]
      ;ENDFOLD
      ;FOLD -- RSK gestartet -- ;%{SE}%MKUKATPVW %CVW_COM %VCOMMENT %P 2:-- RSK gestartet --, 3: VW_COMMENT
      ;ENDFOLD
      ;FOLD F321 = AUS ;%{SE}%MKUKATPVW %CVW_SPS %VBOASG %P 2:F321 = AUS, 3: BOASG
         $FLAG[321] = FALSE
      ;ENDFOLD
      ;FOLD F323 = AUS ;%{SE}%MKUKATPVW %CVW_SPS %VBOASG %P 2:F323 = AUS, 3: BOASG
         $FLAG[323] = FALSE
      ;ENDFOLD
      ;FOLD F324 = AUS ;%{SE}%MKUKATPVW %CVW_SPS %VBOASG %P 2:F324 = AUS, 3: BOASG
         $FLAG[324] = FALSE
      ;ENDFOLD
      ;FOLD F329 = AUS ;%{SE}%MKUKATPVW %CVW_SPS %VBOASG %P 2:F329 = AUS, 3: BOASG
         $FLAG[329] = FALSE
      ;ENDFOLD
      ;FOLD A177 = EIN ;%{SE}%MKUKATPVW %CVW_SPS %VBOASG %P 2:A177 = EIN, 3: BOASG
         $OUT[177] = TRUE
      ;ENDFOLD
      ;FOLD A2123 = AUS ;%{SE}%MKUKATPVW %CVW_SPS %VBOASG %P 2:A2123 = AUS, 3: BOASG
         $OUT[2123] = FALSE
      ;ENDFOLD
      ;FOLD A2124 = AUS ;%{SE}%MKUKATPVW %CVW_SPS %VBOASG %P 2:A2124 = AUS, 3: BOASG
         $OUT[2124] = FALSE
      ;ENDFOLD
      ;FOLD A2125 = AUS ;%{SE}%MKUKATPVW %CVW_SPS %VBOASG %P 2:A2125 = AUS, 3: BOASG
         $OUT[2125] = FALSE
      ;ENDFOLD
      ;FOLD A2126 = AUS ;%{SE}%MKUKATPVW %CVW_SPS %VBOASG %P 2:A2126 = AUS, 3: BOASG
         $OUT[2126] = FALSE
      ;ENDFOLD
      ;FOLD -- Ueberwachungszeit Schwenkeinheit 2 schwenken -- ;%{SE}%MKUKATPVW %CVW_COM %VCOMMENT %P 2:-- Ueberwachungszeit Schwenkeinheit 2 schwenken --, 3: VW_COMMENT
      ;ENDFOLD
      ;FOLD t8 ( EIN ) = -100[1/10Sek] ;%{SE}%MKUKATPVW %CVW_SPS %VTASG %P 2:t8 ( EIN ) = -100[1/10Sek], 3: TASG
         VW(#SET_TIME,TRUE,8,0,-100)
      ;ENDFOLD
      ;FOLD Schritt 201 = !E2123 & A4039  ;%{SE}%MKUKATPVW %CVW_SPS %VST_CON %P 2:Schritt 201 = !E2123 & A4039 , 3: ST_CON
         IF NOT $IN[2123] AND $OUT[4039] THEN
            PREVSTEP = $APP_INT[5]
            $APP_INT[5] = 201
         ENDIF
      ;ENDFOLD
      ;FOLD Schritt 204 = E2123 & !E2124 & A4039  ;%{SE}%MKUKATPVW %CVW_SPS %VST_CON %P 2:Schritt 204 = E2123 & !E2124 & A4039 , 3: ST_CON
         IF $IN[2123] AND NOT $IN[2124] AND $OUT[4039] THEN
            PREVSTEP = $APP_INT[5]
            $APP_INT[5] = 204
         ENDIF
      ;ENDFOLD
   ;ENDFOLD
   ;FOLD SCHRITT 201 --KL2 Spueleimer (an Pneum. Schwenkeinheit KL2)-- ;%{P}%MKUKATPVW,%CSTEP,%VST_NR,%P 1:SCHRITT, 2:201, 3:KL2 Spueleimer (an Pneum. Schwenkeinheit KL2)
      ;FOLD ;%{H}
         Case 201
      ;ENDFOLD
      ;FOLD -- Steuerluft EIN -- ;%{SE}%MKUKATPVW %CVW_COM %VCOMMENT %P 2:-- Steuerluft EIN --, 3: VW_COMMENT
      ;ENDFOLD
      ;FOLD A2121 = A4039 ;%{SE}%MKUKATPVW %CVW_SPS %VBOASG %P 2:A2121 = A4039, 3: BOASG
         $OUT[2121] = $OUT[4039]
      ;ENDFOLD
      ;FOLD -- RSK Fehlerausgabe Schwenkeinheit 2 Arbeit. -- ;%{SE}%MKUKATPVW %CVW_COM %VCOMMENT %P 2:-- RSK Fehlerausgabe Schwenkeinheit 2 Arbeit. --, 3: VW_COMMENT
      ;ENDFOLD
      ;FOLD F324 = !E2124 ;%{SE}%MKUKATPVW %CVW_SPS %VBOASG %P 2:F324 = !E2124, 3: BOASG
         $FLAG[324] = NOT $IN[2124]
      ;ENDFOLD
      ;FOLD -- RSK Sammelstoerung -- ;%{SE}%MKUKATPVW %CVW_COM %VCOMMENT %P 2:-- RSK Sammelstoerung --, 3: VW_COMMENT
      ;ENDFOLD
      ;FOLD F329 = F324 ;%{SE}%MKUKATPVW %CVW_SPS %VBOASG %P 2:F329 = F324, 3: BOASG
         $FLAG[329] = $FLAG[324]
      ;ENDFOLD
      ;FOLD Schritt 200 = (E26 + E27) & F324 & A4039  ;%{SE}%MKUKATPVW %CVW_SPS %VST_CON %P 2:Schritt 200 = (E26 + E27) & F324 & A4039 , 3: ST_CON
         IF ($IN[26] OR $IN[27]) AND $FLAG[324] AND $OUT[4039] THEN
            PREVSTEP = $APP_INT[5]
            $APP_INT[5] = 200
         ENDIF
      ;ENDFOLD
      ;FOLD Schritt 202 = (F523 & !F524 & E2121 + !F523 & F524 & !E2122) & A4039  ;%{SE}%MKUKATPVW %CVW_SPS %VST_CON %P 2:Schritt 202 = (F523 & !F524 & E2121 + !F523 & F524 & !E2122) & A4039 , 3: ST_CON
         IF ($FLAG[523] AND NOT $FLAG[524] AND $IN[2121] OR NOT $FLAG[523] AND $FLAG[524] AND NOT $IN[2122]) AND $OUT[4039] THEN
            PREVSTEP = $APP_INT[5]
            $APP_INT[5] = 202
         ENDIF
      ;ENDFOLD
   ;ENDFOLD
   ;FOLD SCHRITT 202 --KL2 Spueleimer (an Pneum. Schwenkeinheit KL2)-- ;%{P}%MKUKATPVW,%CSTEP,%VST_NR,%P 1:SCHRITT, 2:202, 3:KL2 Spueleimer (an Pneum. Schwenkeinheit KL2)
      ;FOLD ;%{H}
         Case 202
      ;ENDFOLD
      ;FOLD -- Steuerluft EIN -- ;%{SE}%MKUKATPVW %CVW_COM %VCOMMENT %P 2:-- Steuerluft EIN --, 3: VW_COMMENT
      ;ENDFOLD
      ;FOLD A2121 = A4039 ;%{SE}%MKUKATPVW %CVW_SPS %VBOASG %P 2:A2121 = A4039, 3: BOASG
         $OUT[2121] = $OUT[4039]
      ;ENDFOLD
      ;FOLD -- Schwenkeinheit 2 in Ruhestellung schwenken -- ;%{SE}%MKUKATPVW %CVW_COM %VCOMMENT %P 2:-- Schwenkeinheit 2 in Ruhestellung schwenken --, 3: VW_COMMENT
      ;ENDFOLD
      ;FOLD A2123 = EIN ;%{SE}%MKUKATPVW %CVW_SPS %VBOASG %P 2:A2123 = EIN, 3: BOASG
         $OUT[2123] = TRUE
      ;ENDFOLD
      ;FOLD A2124 = AUS ;%{SE}%MKUKATPVW %CVW_SPS %VBOASG %P 2:A2124 = AUS, 3: BOASG
         $OUT[2124] = FALSE
      ;ENDFOLD
      ;FOLD -- FRG Bewegung EIN -- ;%{SE}%MKUKATPVW %CVW_COM %VCOMMENT %P 2:-- FRG Bewegung EIN --, 3: VW_COMMENT
      ;ENDFOLD
      ;FOLD A2125 = AUS ;%{SE}%MKUKATPVW %CVW_SPS %VBOASG %P 2:A2125 = AUS, 3: BOASG
         $OUT[2125] = FALSE
      ;ENDFOLD
      ;FOLD A2126 = EIN ;%{SE}%MKUKATPVW %CVW_SPS %VBOASG %P 2:A2126 = EIN, 3: BOASG
         $OUT[2126] = TRUE
      ;ENDFOLD
      ;FOLD Schritt 203 = !E2124 & E2123 & A4039 + T8  ;%{SE}%MKUKATPVW %CVW_SPS %VST_CON %P 2:Schritt 203 = !E2124 & E2123 & A4039 + T8 , 3: ST_CON
         IF NOT $IN[2124] AND $IN[2123] AND $OUT[4039] OR $TIMER_FLAG[8] THEN
            PREVSTEP = $APP_INT[5]
            $APP_INT[5] = 203
         ENDIF
      ;ENDFOLD
   ;ENDFOLD
   ;FOLD SCHRITT 203 --KL2 Spueleimer (an Pneum. Schwenkeinheit KL2)-- ;%{P}%MKUKATPVW,%CSTEP,%VST_NR,%P 1:SCHRITT, 2:203, 3:KL2 Spueleimer (an Pneum. Schwenkeinheit KL2)
      ;FOLD ;%{H}
         Case 203
      ;ENDFOLD
      ;FOLD -- Steuerluft EIN -- ;%{SE}%MKUKATPVW %CVW_COM %VCOMMENT %P 2:-- Steuerluft EIN --, 3: VW_COMMENT
      ;ENDFOLD
      ;FOLD A2121 = A4039 ;%{SE}%MKUKATPVW %CVW_SPS %VBOASG %P 2:A2121 = A4039, 3: BOASG
         $OUT[2121] = $OUT[4039]
      ;ENDFOLD
      ;FOLD -- RSK Fehlerausgabe Schwenkeinheit 2 Ruhestellung -- ;%{SE}%MKUKATPVW %CVW_COM %VCOMMENT %P 2:-- RSK Fehlerausgabe Schwenkeinheit 2 Ruhestellung --, 3: VW_COMMENT
      ;ENDFOLD
      ;FOLD F323 = !E2123 & T8 + F323 ;%{SE}%MKUKATPVW %CVW_SPS %VBOASG %P 2:F323 = !E2123 & T8 + F323, 3: BOASG
         $FLAG[323] = NOT $IN[2123] AND $TIMER_FLAG[8] OR $FLAG[323]
      ;ENDFOLD
      ;FOLD -- RSK Sammelstoerung -- ;%{SE}%MKUKATPVW %CVW_COM %VCOMMENT %P 2:-- RSK Sammelstoerung --, 3: VW_COMMENT
      ;ENDFOLD
      ;FOLD F329 = F323 ;%{SE}%MKUKATPVW %CVW_SPS %VBOASG %P 2:F329 = F323, 3: BOASG
         $FLAG[329] = $FLAG[323]
      ;ENDFOLD
      ;FOLD A2123 = AUS ;%{SE}%MKUKATPVW %CVW_SPS %VBOASG %P 2:A2123 = AUS, 3: BOASG
         $OUT[2123] = FALSE
      ;ENDFOLD
      ;FOLD -- FRG Bewegung AUS -- ;%{SE}%MKUKATPVW %CVW_COM %VCOMMENT %P 2:-- FRG Bewegung AUS --, 3: VW_COMMENT
      ;ENDFOLD
      ;FOLD A2126 = AUS ;%{SE}%MKUKATPVW %CVW_SPS %VBOASG %P 2:A2126 = AUS, 3: BOASG
         $OUT[2126] = FALSE
      ;ENDFOLD
      ;FOLD Schritt 200 = F323 & (E26 + E27) & A4039  ;%{SE}%MKUKATPVW %CVW_SPS %VST_CON %P 2:Schritt 200 = F323 & (E26 + E27) & A4039 , 3: ST_CON
         IF $FLAG[323] AND ($IN[26] OR $IN[27]) AND $OUT[4039] THEN
            PREVSTEP = $APP_INT[5]
            $APP_INT[5] = 200
         ENDIF
      ;ENDFOLD
      ;FOLD Schritt 204 = !F323 & (E2126 + F837) & A4039  ;%{SE}%MKUKATPVW %CVW_SPS %VST_CON %P 2:Schritt 204 = !F323 & (E2126 + F837) & A4039 , 3: ST_CON
         IF NOT $FLAG[323] AND ($IN[2126] OR $FLAG[837]) AND $OUT[4039] THEN
            PREVSTEP = $APP_INT[5]
            $APP_INT[5] = 204
         ENDIF
      ;ENDFOLD
   ;ENDFOLD
   ;FOLD SCHRITT 204 --KL2 Spueleimer (an Pneum. Schwenkeinheit KL2)-- ;%{P}%MKUKATPVW,%CSTEP,%VST_NR,%P 1:SCHRITT, 2:204, 3:KL2 Spueleimer (an Pneum. Schwenkeinheit KL2)
      ;FOLD ;%{H}
         Case 204
      ;ENDFOLD
      ;FOLD -- Steuerluft EIN -- ;%{SE}%MKUKATPVW %CVW_COM %VCOMMENT %P 2:-- Steuerluft EIN --, 3: VW_COMMENT
      ;ENDFOLD
      ;FOLD A2121 = A4039 ;%{SE}%MKUKATPVW %CVW_SPS %VBOASG %P 2:A2121 = A4039, 3: BOASG
         $OUT[2121] = $OUT[4039]
      ;ENDFOLD
      ;FOLD F323 = AUS ;%{SE}%MKUKATPVW %CVW_SPS %VBOASG %P 2:F323 = AUS, 3: BOASG
         $FLAG[323] = FALSE
      ;ENDFOLD
      ;FOLD F329 = T8 ;%{SE}%MKUKATPVW %CVW_SPS %VBOASG %P 2:F329 = T8, 3: BOASG
         $FLAG[329] = $TIMER_FLAG[8]
      ;ENDFOLD
      ;FOLD -- FRG in Endlage halten ein -- ;%{SE}%MKUKATPVW %CVW_COM %VCOMMENT %P 2:-- FRG in Endlage halten ein --, 3: VW_COMMENT
      ;ENDFOLD
      ;FOLD A2125 = EIN ;%{SE}%MKUKATPVW %CVW_SPS %VBOASG %P 2:A2125 = EIN, 3: BOASG
         $OUT[2125] = TRUE
      ;ENDFOLD
      ;FOLD Schritt 205 = !E2125 & (E2126 + F837) & A4039  ;%{SE}%MKUKATPVW %CVW_SPS %VST_CON %P 2:Schritt 205 = !E2125 & (E2126 + F837) & A4039 , 3: ST_CON
         IF NOT $IN[2125] AND ($IN[2126] OR $FLAG[837]) AND $OUT[4039] THEN
            PREVSTEP = $APP_INT[5]
            $APP_INT[5] = 205
         ENDIF
      ;ENDFOLD
   ;ENDFOLD
   ;FOLD SCHRITT 205 --KL2 Spueleimer (an Pneum. Schwenkeinheit KL2)-- ;%{P}%MKUKATPVW,%CSTEP,%VST_NR,%P 1:SCHRITT, 2:205, 3:KL2 Spueleimer (an Pneum. Schwenkeinheit KL2)
      ;FOLD ;%{H}
         Case 205
      ;ENDFOLD
      ;FOLD -- Steuerluft EIN -- ;%{SE}%MKUKATPVW %CVW_COM %VCOMMENT %P 2:-- Steuerluft EIN --, 3: VW_COMMENT
      ;ENDFOLD
      ;FOLD A2121 = A4039 ;%{SE}%MKUKATPVW %CVW_SPS %VBOASG %P 2:A2121 = A4039, 3: BOASG
         $OUT[2121] = $OUT[4039]
      ;ENDFOLD
      ;FOLD -- RSK Sammelstoerung -- ;%{SE}%MKUKATPVW %CVW_COM %VCOMMENT %P 2:-- RSK Sammelstoerung --, 3: VW_COMMENT
      ;ENDFOLD
      ;FOLD F329 = T8 ;%{SE}%MKUKATPVW %CVW_SPS %VBOASG %P 2:F329 = T8, 3: BOASG
         $FLAG[329] = $TIMER_FLAG[8]
      ;ENDFOLD
      ;FOLD -- FRG in Endlage halten AUS -- ;%{SE}%MKUKATPVW %CVW_COM %VCOMMENT %P 2:-- FRG in Endlage halten AUS --, 3: VW_COMMENT
      ;ENDFOLD
      ;FOLD A2125 = AUS ;%{SE}%MKUKATPVW %CVW_SPS %VBOASG %P 2:A2125 = AUS, 3: BOASG
         $OUT[2125] = FALSE
      ;ENDFOLD
      ;FOLD A177 = AUS ;%{SE}%MKUKATPVW %CVW_SPS %VBOASG %P 2:A177 = AUS, 3: BOASG
         $OUT[177] = FALSE
      ;ENDFOLD
      ;FOLD t8 ( EIN ) = STOP ;%{SE}%MKUKATPVW %CVW_SPS %VTSTOP %P 2:t8 ( EIN ) = STOP, 3: TSTOP
         VW(#SET_TIME,TRUE,8,1,0)
      ;ENDFOLD
      ;FOLD F376 =  E2123 & !E2124 ;%{SE}%MKUKATPVW %CVW_SPS %VBOASG %P 2:F376 =  E2123 & !E2124, 3: BOASG
         $FLAG[376] = $IN[2123] AND NOT $IN[2124]
      ;ENDFOLD
      ;FOLD Schritt 1 = F376 & A4039  ;%{SE}%MKUKATPVW %CVW_SPS %VST_CON %P 2:Schritt 1 = F376 & A4039 , 3: ST_CON
         IF $FLAG[376] AND $OUT[4039] THEN
            PREVSTEP = $APP_INT[5]
            $APP_INT[5] = 1
         ENDIF
      ;ENDFOLD
   ;ENDFOLD
   ;FOLD SCHRITT 206 --KL3 Spueleimer (an Pneum. Schwenkeinheit KL3)-- ;%{P}%MKUKATPVW,%CSTEP,%VST_NR,%P 1:SCHRITT, 2:206, 3:KL3 Spueleimer (an Pneum. Schwenkeinheit KL3)
      ;FOLD ;%{H}
         Case 206
      ;ENDFOLD
      ;FOLD -- RSK gestartet -- ;%{SE}%MKUKATPVW %CVW_COM %VCOMMENT %P 2:-- RSK gestartet --, 3: VW_COMMENT
      ;ENDFOLD
      ;FOLD F321 = AUS ;%{SE}%MKUKATPVW %CVW_SPS %VBOASG %P 2:F321 = AUS, 3: BOASG
         $FLAG[321] = FALSE
      ;ENDFOLD
      ;FOLD F323 = AUS ;%{SE}%MKUKATPVW %CVW_SPS %VBOASG %P 2:F323 = AUS, 3: BOASG
         $FLAG[323] = FALSE
      ;ENDFOLD
      ;FOLD F324 = AUS ;%{SE}%MKUKATPVW %CVW_SPS %VBOASG %P 2:F324 = AUS, 3: BOASG
         $FLAG[324] = FALSE
      ;ENDFOLD
      ;FOLD F329 = AUS ;%{SE}%MKUKATPVW %CVW_SPS %VBOASG %P 2:F329 = AUS, 3: BOASG
         $FLAG[329] = FALSE
      ;ENDFOLD
      ;FOLD A193 = EIN ;%{SE}%MKUKATPVW %CVW_SPS %VBOASG %P 2:A193 = EIN, 3: BOASG
         $OUT[193] = TRUE
      ;ENDFOLD
      ;FOLD -- Steuerluft EIN -- ;%{SE}%MKUKATPVW %CVW_COM %VCOMMENT %P 2:-- Steuerluft EIN --, 3: VW_COMMENT
      ;ENDFOLD
      ;FOLD A2129 = A4039 ;%{SE}%MKUKATPVW %CVW_SPS %VBOASG %P 2:A2129 = A4039, 3: BOASG
         $OUT[2129] = $OUT[4039]
      ;ENDFOLD
      ;FOLD A2131 = AUS ;%{SE}%MKUKATPVW %CVW_SPS %VBOASG %P 2:A2131 = AUS, 3: BOASG
         $OUT[2131] = FALSE
      ;ENDFOLD
      ;FOLD A2132 = AUS ;%{SE}%MKUKATPVW %CVW_SPS %VBOASG %P 2:A2132 = AUS, 3: BOASG
         $OUT[2132] = FALSE
      ;ENDFOLD
      ;FOLD A2133 = AUS ;%{SE}%MKUKATPVW %CVW_SPS %VBOASG %P 2:A2133 = AUS, 3: BOASG
         $OUT[2133] = FALSE
      ;ENDFOLD
      ;FOLD A2134 = AUS ;%{SE}%MKUKATPVW %CVW_SPS %VBOASG %P 2:A2134 = AUS, 3: BOASG
         $OUT[2134] = FALSE
      ;ENDFOLD
      ;FOLD -- Ueberwachungszeit Schwenkeinheit 3 -- ;%{SE}%MKUKATPVW %CVW_COM %VCOMMENT %P 2:-- Ueberwachungszeit Schwenkeinheit 3 --, 3: VW_COMMENT
      ;ENDFOLD
      ;FOLD t8 ( EIN ) = -100[1/10Sek] ;%{SE}%MKUKATPVW %CVW_SPS %VTASG %P 2:t8 ( EIN ) = -100[1/10Sek], 3: TASG
         VW(#SET_TIME,TRUE,8,0,-100)
      ;ENDFOLD
